# B&R Automation Studio project CombinedLinenCleanA6 (part 7)

#### _SetCAN2TypeToCAN1Type.ab
```automation-basic
FUNCTION_BLOCK _SetCAN2TypeToCAN1Type
;********************************************************************************************************
; * Implementation of _SetCAN2TypeToCAN1Type
;********************************************************************************************************
; * version 		1.10
;	* ###HO - 020905 - Fünftes Telegramm ergänzt
; * version 		1.00
; * last change		sep, 30th, 2003
; * by				H.O.
;********************************************************************************************************
;********************************************************************************************************
; 	-> 	pCAN2Data			.. pointer to CAN2 structure that contains data to read or write
; 	-> 	iTelegramIndex		.. telegram index exctractet from received / broadcasted telegram
; 		pCAN1Data 		->	.. return the address of CAN1 struct
;********************************************************************************************************

; set local pointer to incoming CAN2 uni structure
memcpy(adr(LocalCAN2UniData), pCAN2Data, sizeof(LocalCAN2UniData))

iStatus = 0

; create CAN1 telegram from CAN2 te structure passed in..
case iTelegramIndex of
	action 1:
		LocalCAN1Data.T_By0 	= LocalCAN2UniData.T1_By0
		LocalCAN1Data.T_By1 	= LocalCAN2UniData.T1_By1
		LocalCAN1Data.T_By2_By3 = LocalCAN2UniData.T1_By2_By3
		LocalCAN1Data.T_By4_By5 = LocalCAN2UniData.T1_By4_By5
		LocalCAN1Data.T_By6_By7 = LocalCAN2UniData.T1_By6_By7
	endaction
	action 2:
		LocalCAN1Data.T_By0 	= LocalCAN2UniData.T2_By0
		LocalCAN1Data.T_By1 	= LocalCAN2UniData.T2_By1
		LocalCAN1Data.T_By2_By3 = LocalCAN2UniData.T2_By2_By3
		LocalCAN1Data.T_By4_By5 = LocalCAN2UniData.T2_By4_By5
		LocalCAN1Data.T_By6_By7 = LocalCAN2UniData.T2_By6_By7
	endaction
	action 3:
		LocalCAN1Data.T_By0 	= LocalCAN2UniData.T3_By0
		LocalCAN1Data.T_By1 	= LocalCAN2UniData.T3_By1
		LocalCAN1Data.T_By2_By3 = LocalCAN2UniData.T3_By2_By3
		LocalCAN1Data.T_By4_By5 = LocalCAN2UniData.T3_By4_By5
		LocalCAN1Data.T_By6_By7 = LocalCAN2UniData.T3_By6_By7
	endaction
	action 4:
		LocalCAN1Data.T_By0 	= LocalCAN2UniData.T4_By0
		LocalCAN1Data.T_By1 	= LocalCAN2UniData.T4_By1
		LocalCAN1Data.T_By2_By3 = LocalCAN2UniData.T4_By2_By3
		LocalCAN1Data.T_By4_By5 = LocalCAN2UniData.T4_By4_By5
		LocalCAN1Data.T_By6_By7 = LocalCAN2UniData.T4_By6_By7
	endaction
	action 5:
		LocalCAN1Data.T_By0 	= LocalCAN2UniData.T5_By0
		LocalCAN1Data.T_By1 	= LocalCAN2UniData.T5_By1
		LocalCAN1Data.T_By2_By3 = LocalCAN2UniData.T5_By2_By3
		LocalCAN1Data.T_By4_By5 = LocalCAN2UniData.T5_By4_By5
		LocalCAN1Data.T_By6_By7 = LocalCAN2UniData.T5_By6_By7
	endaction
	elseaction:
		iStatus = 109
	endaction
endcase

; pass pointer to CAN1 telegram to output..
pCAN1Data = ADR(LocalCAN1Data)

;********************************************************************************************************
;********************************************************************************************************
END_FUNCTION_BLOCK
```

#### _GetCANIDFromObjNr.ab
```automation-basic
FUNCTION_BLOCK _GetCANIDFromObjNr
;********************************************************************************************************
; * Implementation of _GetCANIDFromObjNr
;********************************************************************************************************
; * version 		3.6.0
; * last change		120210
; * by				H.O.
;********************************************************************************************************
; History:
;*********
; V3.6.0 - ###HO - 120210
;	* COB120 auch für ID 150,160,170,180,190
;	* COB121 auch für ID 151,161,171,181,191
; * V3.4.0 ###HO
; 	- COB ID 110 + 111
; * V3.2.1 ###HO
; 	- COB 130,140 wie 120  und...
;	- 131 und 141 wie 121
; * V3.2.0 ###HO  - 040907
;  	* COBs 261+262 hinzugefügt
; 	* COBs302,303,304,312,313,314,253,255,254,256,352,353,354  neu
;	* udCANID = udObjNr für alle erwähnten Objektnummern
; * V3.1.0 ###HO  - 141206
; 	* COBs 126,127,128,129 hinzugefügt
; * V3.0.0 ###HO  - 120905
; 	* IDs 253..258 hinzugefügt
; 	* IDs 307..317 hinzugefügt
; * V 1.0.0  	* Erste Version
; * V 2.0.0 HO 	* COBs 251,252,480,481 added
; 				* COB 123 added
; * V2.1.0 HO	* COB 441..459 added
;********************************************************************************************************
; supported CANIDs: 120,121,122,123,130,140,131,141,201,209,211,219,221,231,251,252
; 					301,306,311,316,351,361..369,371..379,401..419,421..439,441..459,480,481
;********************************************************************************************************

; ObjNr and CANID are identical..
iStatus = 0
case udObjNr of

    action 120 :
    action 126 :
    action 128 :
    action 130 :
    action 140 :
	action 150:
	action 160:
	action 170:
	action 180:
	action 190:
        udCANID = 120
    endaction
   	action 121:
    action 127 :
    action 129 :
    action 131 :
    action 141 :
	action 151:
	action 161:
	action 171:
	action 181:
	action 191:
        udCANID = 121
	endaction

	action 110 :
	action 111 :
	action 122 :
   	action 123 :
	action 201:
	action 209:
	action 211:
	action 219:
	action 221:
	action 231:
	action 251:
	action 252:
	action 253:
	action 254:
	action 255:
	action 256:
	action 257:
	action 258:
	action 261:
	action 262:
	action 301:
	action 302:
	action 303:
	action 304:
	action 306:
	action 307:
	action 311:
	action 312:
	action 313:
	action 314:
	action 316:
	action 317:
	action 351:
	action 352:
	action 353:
	action 354:
	action 361..369:
	action 371..379:
	action 401..419:
	action 421..439:
	action 441..459:
	action 480:
	action 481:
        udCANID = udObjNr
	endaction
	elseaction:
		; all other ObjNrs..
		iStatus = 110
	endaction
endcase
;********************************************************************************************************
END_FUNCTION_BLOCK
```

#### _GetPVSize.ab
```automation-basic
FUNCTION_BLOCK _GetPVSize
;********************************************************************************************************
; * Implementation of _GetPVSize
;********************************************************************************************************
; * version 		3.6.0
; * last change		120210
; * by				H.O.
;********************************************************************************************************
; History:
;*********
; V3.6.0 - ###HO - 120210
;	* COB120 auch für ID 150,160,170,180,190
;	* COB121 auch für ID 151,161,171,181,191
; * V3.4.0
;	* COB ID 110 + 111
; * V3.2.1
;	* COB130,140 wie 120 und..
;	* COB 131,141 wie 121
; * V3.2.0
; 	* COBs 261,262 hinzugefügt
; 	* COBs302,303,304,312,313,314,253,255,254,256,352,353,354  neu
; 	* gleiche Objekte durch MehrfachAction zusammengefasst
; * V3.1.0
; 	* COBs 126,127,128,129,130 hinzugefügt
; * V3.0.0
; 	* COBs 253..258 -> gleiche Strukturen mit anderen IDs (hcs)
; * V 1.0.0 	-> Original
; * V 2.0.0 HO 	* COBs 251,252,480,481 added
;				* COB 123 added
; * V2.1.0	HO	* COB441..459 added

;********************************************************************************************************
; supported CANIDs: 120,121,122,123,130,140,131,141,201,209,211,219,221,231,251,252
; 					301,306,311,316,351,361..369,371..379,401..419,421..439,441bis459,480,481
;********************************************************************************************************

iStatus = 0
case uiObjNr of
action 110:
	iCobLength = sizeof (COB_Typ_110)
endaction
action 111:
	iCobLength = sizeof (COB_Typ_111)
endaction
action 120:
action 126:
action 128:
action 130:
action 140:
action 150:
action 160:
action 170:
action 180:
action 190:
	iCobLength = sizeof (COBTyp_120)
endaction
action 121:
action 127:
action 129:
action 131:
action 141:
action 151:
action 161:
action 171:
action 181:
action 191:
	iCobLength = sizeof (COBTyp_121)
endaction
action 122:
	iCobLength = sizeof (COBTyp_122)
endaction
action 123:
	iCobLength = sizeof (COBTyp_123)
endaction
(*
action 1130:	; 08.10.2007 - (hcs) DEAKTIVIERT
	iCobLength = sizeof (COB_Typ_130_140)
endaction
action 1131:	; 08.10.2007 - (hcs) DEAKTIVIERT
  	iCobLength = sizeof (COB_Typ_131_141)
endaction
action 140:
	iCobLength = sizeof (COB_Typ_130_140)
endaction
action 141:
  	iCobLength = sizeof (COB_Typ_131_141)
endaction
*)
action 201:
   	iCobLength = sizeof (COB_Typ_201)
endaction
action 209:
   	iCobLength = sizeof (COB_Typ_209)
endaction
action 211:
   	iCobLength = sizeof (COB_Typ_211)
endaction
action 219:
   	iCobLength = sizeof (COB_Typ_219)
endaction
action 221:
	iCobLength = sizeof (COB_Typ_221)
endaction
action 231:
	iCobLength = sizeof (COB_Typ_231)
endaction
action 251:
action 253:
action 255:
action 257:
	iCobLength = sizeof (COBTyp_251)
endaction
action 252:
action 254:
action 256:
action 258:
	iCobLength = sizeof (COBTyp_252)
endaction
action 261:
	iCobLength = sizeof (COB_Typ_261)
endaction
action 262:
	iCobLength = sizeof (COB_Typ_262)
endaction
action 301:
action 302:
action 303:
action 304:
	iCobLength = sizeof (COB_Typ_301)
endaction
action 306:
	iCobLength = sizeof (COB_Typ_306)
endaction
action 307:
	iCobLength = sizeof (COB_Typ_307)
endaction
action 311:
action 312:
action 313:
action 314:
	iCobLength = sizeof (COB_Typ_311)
endaction
action 316:
	iCobLength = sizeof (COB_Typ_316)
endaction
action 317:
	iCobLength = sizeof (COB_Typ_317)
endaction
action 351:
action 352:
action 353:
action 354:
	iCobLength = sizeof (COB_Typ_351)
endaction
action 361..369:
	iCobLength = sizeof (COB_Typ_361bis369)
endaction
action 371..379:
	iCobLength = sizeof (COB_Typ_371bis379)
endaction
action 401..419:
	iCobLength = sizeof (COB_Typ_401bis419)
endaction
action 421..439:
	iCobLength = sizeof (COB_Typ_421bis439)
endaction
action 441..459:
	iCobLength = sizeof (COB_Typ_441bis459)
endaction
action 480:
	iCobLength = sizeof (COBTyp_480)
endaction
action 481:
	iCobLength = sizeof (COBTyp_481)
endaction

; all other ObjNrs..
elseaction:
	iStatus = 110
endaction

endcase
;********************************************************************************************************
END_FUNCTION_BLOCK
```

#### _ConvertDataToi386.ab
```automation-basic
FUNCTION_BLOCK _ConvertDataToi386
;********************************************************************************************************
; * Implementation of _ConvertDataToi386
; 	*** Only ReadOperation for IntelTarget***
;********************************************************************************************************
; * version 		3.6.0
; * last change		120210
; * by				H.O.
;********************************************************************************************************
; History:
; --------
; V3.6.0 - ###HO - 120210
;	* COB120 auch für ID 150,160,170,180,190
;	* COB121 auch für ID 151,161,171,181,191
; * V3.4.0
;	* COB ID 110 + 111
; * V3.2.1
;	* COB130,140 wie 120 und..
;	* COB 131,141 wie 121
; * V3.2.0 HO 040907
;	* _ConvertDataToi386.COB251.bStartBeladung
;	* COBs 261,262 added
; 	* COBs302,303,304,312,313,314,253,255,254,256,352,353,354  neu
; * V3.1.0 HO 141206
;	* COBs 126,127,128,129 hinzugefügt
; * V3.0.0 HO 070905
;		cob251
; * V2.1.0 HO 150404
;		* Redundancy support done for COBs: 480,481
; * V 2.0.0 (by HO) -> COBs 251,252,480,481 added
; 					-> COBs 120,121,123 modified
; 					-> COB 122 replaced
; * V 1.0.0  		-> Original
;********************************************************************************************************
; this function transforms an incoming ByteArray in motorola order to intel format:
;  -> performs address adaption to intel format
; 		(intel requires swapping of WORDs and modification of startadresses by DWORDs (dividable by four))
;  -> swapping of single WORDS of LONG
;  -> swapping of single WORDS (= uints) is not necessary
;  -> swapping of neighboring characters of STRING
;********************************************************************************************************
; supported CANIDs: 120, 121,122,123,130,140,131,141,201,209,211,219,221,231,251,252
; 					301,306,311,316,351,361..369,371..379,401..419,421..439,480,481
;********************************************************************************************************

; always assign InData to OutData -> overwrite changes..
ByteArrayi386 = ByteArrayMotorola

case uiObjNr of
	action 120:
	action 126:
	action 128:
	action 130:
	action 140:
	action 150:
	action 160:
	action 170:
	action 180:
	action 190:
		; udPostennummer
		ByteArrayi386[8] 	= ByteArrayMotorola[10]
		ByteArrayi386[9] 	= ByteArrayMotorola[11]
		ByteArrayi386[10] 	= ByteArrayMotorola[8]
		ByteArrayi386[11] 	= ByteArrayMotorola[9]

		; szAuftragskennzeichen
		usTempByte 			= ByteArrayMotorola[14]
		ByteArrayi386[14] 	= ByteArrayMotorola[15]
		ByteArrayi386[15] 	= usTempByte
		usTempByte 			= ByteArrayMotorola[16]
		ByteArrayi386[16] 	= ByteArrayMotorola[17]
		ByteArrayi386[17] 	= usTempByte
		usTempByte 			= ByteArrayMotorola[18]
		ByteArrayi386[18] 	= ByteArrayMotorola[19]
		ByteArrayi386[19] 	= usTempByte
		usTempByte 			= ByteArrayMotorola[20]
		ByteArrayi386[20] 	= ByteArrayMotorola[21]
		ByteArrayi386[21] 	= usTempByte
		usTempByte 			= ByteArrayMotorola[22]
		ByteArrayi386[22] 	= ByteArrayMotorola[23]
		ByteArrayi386[23] 	= usTempByte
		usTempByte 			= ByteArrayMotorola[24]
		ByteArrayi386[24] 	= ByteArrayMotorola[25]
		ByteArrayi386[25] 	= usTempByte
		; + EOS +  Alignment

		; ud Kundennummer
		ByteArrayi386[28] 	= ByteArrayMotorola[30]
		ByteArrayi386[29] 	= ByteArrayMotorola[31]
		ByteArrayi386[30] 	= ByteArrayMotorola[28]
		ByteArrayi386[31] 	= ByteArrayMotorola[29]

	endaction ; 120

	action 121:
	action 127:
	action 129:
	action 131:
	action 141:
	action 151:
	action 161:
	action 171:
	action 181:
	action 191:
		; nothing to do..
	endaction ; 121

	; replaced from V2.0.0
	action 122:
		; udKundennummer
		ByteArrayi386[4] 	= ByteArrayMotorola[6]
		ByteArrayi386[5] 	= ByteArrayMotorola[7]
		ByteArrayi386[6] 	= ByteArrayMotorola[4]
		ByteArrayi386[7] 	= ByteArrayMotorola[5]

		; udPostennummer
		ByteArrayi386[12] 	= ByteArrayMotorola[14]
		ByteArrayi386[13] 	= ByteArrayMotorola[15]
		ByteArrayi386[14] 	= ByteArrayMotorola[12]
		ByteArrayi386[15] 	= ByteArrayMotorola[13]

		; szAuftragskennzeichen
		usTempByte 			= ByteArrayMotorola[17]
		ByteArrayi386[17] 	= ByteArrayMotorola[18]
		ByteArrayi386[18] 	= usTempByte
		usTempByte 			= ByteArrayMotorola[19]
		ByteArrayi386[19] 	= ByteArrayMotorola[20]
		ByteArrayi386[20] 	= usTempByte
		usTempByte 			= ByteArrayMotorola[21]
		ByteArrayi386[21] 	= ByteArrayMotorola[22]
		ByteArrayi386[22] 	= usTempByte
		usTempByte 			= ByteArrayMotorola[23]
		ByteArrayi386[23] 	= ByteArrayMotorola[24]
		ByteArrayi386[24] 	= usTempByte
		usTempByte 			= ByteArrayMotorola[25]
		ByteArrayi386[25] 	= ByteArrayMotorola[26]
		ByteArrayi386[26] 	= usTempByte
		usTempByte 			= ByteArrayMotorola[27]
		ByteArrayi386[27] 	= ByteArrayMotorola[28]
		ByteArrayi386[28] 	= usTempByte
	endaction ; 122

	action 123:
		; nothing to do..
	endaction ; 123
(*
	action 1130: 			; 08.10.2007 - (hcs) DEAKTIVIERT
		; udPostennummer
		ByteArrayi386[12] 	= ByteArrayMotorola[12]
		ByteArrayi386[13] 	= ByteArrayMotorola[13]
		ByteArrayi386[14] 	= ByteArrayMotorola[10]
		ByteArrayi386[15] 	= ByteArrayMotorola[11]

		; usFehlernummer
		ByteArrayi386[16] 	= ByteArrayMotorola[14]

		; bAuftragskennzeichen
		ByteArrayi386[17] 	= ByteArrayMotorola[15]

		; szAuftragskennzeichen
			ByteArrayi386[18] 	= ByteArrayMotorola[17]
		ByteArrayi386[19] 	= ByteArrayMotorola[16]
			ByteArrayi386[20] 	= ByteArrayMotorola[19]
		ByteArrayi386[21] 	= ByteArrayMotorola[18]
			ByteArrayi386[22] 	= ByteArrayMotorola[21]
		ByteArrayi386[23] 	= ByteArrayMotorola[20]
			ByteArrayi386[24] 	= ByteArrayMotorola[23]
		ByteArrayi386[25] 	= ByteArrayMotorola[22]
			ByteArrayi386[26] 	= ByteArrayMotorola[25]
		ByteArrayi386[27] 	= ByteArrayMotorola[24]
			ByteArrayi386[28] 	= ByteArrayMotorola[27]
		ByteArrayi386[29] 	= ByteArrayMotorola[26]

		; udKundennummer
		ByteArrayi386[32] 	= ByteArrayMotorola[32]
		ByteArrayi386[33] 	= ByteArrayMotorola[33]
		ByteArrayi386[34] 	= ByteArrayMotorola[30]
		ByteArrayi386[35] 	= ByteArrayMotorola[31]

		; uiGewicht
		ByteArrayi386[36] 	= ByteArrayMotorola[34]
		ByteArrayi386[37] 	= ByteArrayMotorola[35]

		; bNotAusEnts
		ByteArrayi386[38] 	= ByteArrayMotorola[36]
	endaction ; 130

	action 140:
		; udPostennummer
		ByteArrayi386[12] 	= ByteArrayMotorola[12]
		ByteArrayi386[13] 	= ByteArrayMotorola[13]
		ByteArrayi386[14] 	= ByteArrayMotorola[10]
		ByteArrayi386[15] 	= ByteArrayMotorola[11]

		; usFehlernummer
		ByteArrayi386[16] 	= ByteArrayMotorola[14]

		; bAuftragskennzeichen
		ByteArrayi386[17] 	= ByteArrayMotorola[15]

		; szAuftragskennzeichen
			ByteArrayi386[18] 	= ByteArrayMotorola[17]
		ByteArrayi386[19] 	= ByteArrayMotorola[16]
			ByteArrayi386[20] 	= ByteArrayMotorola[19]
		ByteArrayi386[21] 	= ByteArrayMotorola[18]
			ByteArrayi386[22] 	= ByteArrayMotorola[21]
		ByteArrayi386[23] 	= ByteArrayMotorola[20]
			ByteArrayi386[24] 	= ByteArrayMotorola[23]
		ByteArrayi386[25] 	= ByteArrayMotorola[22]
			ByteArrayi386[26] 	= ByteArrayMotorola[25]
		ByteArrayi386[27] 	= ByteArrayMotorola[24]
			ByteArrayi386[28] 	= ByteArrayMotorola[27]
		ByteArrayi386[29] 	= ByteArrayMotorola[26]

		; udKundennummer
		ByteArrayi386[32] 	= ByteArrayMotorola[32]
		ByteArrayi386[33] 	= ByteArrayMotorola[33]
		ByteArrayi386[34] 	= ByteArrayMotorola[30]
		ByteArrayi386[35] 	= ByteArrayMotorola[31]

		; uiGewicht
		ByteArrayi386[36] 	= ByteArrayMotorola[34]
		ByteArrayi386[37] 	= ByteArrayMotorola[35]

		; bNotAusEnts
		ByteArrayi386[38] 	= ByteArrayMotorola[36]
	endaction ; 140

	action 1131: 	; 08.10.2007 - (hcs) DEAKTIVIERT
		; nothing to do
	endaction ; 131..141

	action 141:
		; nothing to do
	endaction ; 131..141
*)
	action 201:
	; nur swappen - kein Alignment
		; udPostennummer
		ByteArrayi386[8] 	= ByteArrayMotorola[10]
		ByteArrayi386[9] 	= ByteArrayMotorola[11]
		ByteArrayi386[10] 	= ByteArrayMotorola[8]
		ByteArrayi386[11] 	= ByteArrayMotorola[9]

		; udKundennummer
		ByteArrayi386[12] 	= ByteArrayMotorola[14]
		ByteArrayi386[13] 	= ByteArrayMotorola[15]
		ByteArrayi386[14] 	= ByteArrayMotorola[12]
		ByteArrayi386[15] 	= ByteArrayMotorola[13]
	endaction ; 201

	action 209:
		; udPostennummer
		ByteArrayi386[8] 	= ByteArrayMotorola[10]
		ByteArrayi386[9] 	= ByteArrayMotorola[11]
		ByteArrayi386[10] 	= ByteArrayMotorola[8]
		ByteArrayi386[11] 	= ByteArrayMotorola[9]

		; udKundennummer
		ByteArrayi386[12] 	= ByteArrayMotorola[14]
		ByteArrayi386[13] 	= ByteArrayMotorola[15]
		ByteArrayi386[14] 	= ByteArrayMotorola[12]
		ByteArrayi386[15] 	= ByteArrayMotorola[13]
	endaction ; 209

	action 211:
		; nothing to do
	endaction ; 211

	action 219:
		; nothing to do
		ByteArrayi386[6] 	= ByteArrayMotorola[7]
		ByteArrayi386[7] 	= ByteArrayMotorola[6]
	endaction ; 219

	action 221:
		; udPostennummer
		ByteArrayi386[8] 	= ByteArrayMotorola[8]
		ByteArrayi386[9] 	= ByteArrayMotorola[9]
		ByteArrayi386[10] 	= ByteArrayMotorola[6]
		ByteArrayi386[11] 	= ByteArrayMotorola[7]
		; udKundennummer
		ByteArrayi386[12] 	= ByteArrayMotorola[12]
		ByteArrayi386[13] 	= ByteArrayMotorola[13]
		ByteArrayi386[14] 	= ByteArrayMotorola[10]
		ByteArrayi386[15] 	= ByteArrayMotorola[11]
		; uiGewicht
		ByteArrayi386[16] 	= ByteArrayMotorola[14]
		ByteArrayi386[17] 	= ByteArrayMotorola[15]
		; bNotAusWM
		ByteArrayi386[18] 	= ByteArrayMotorola[16]
		; Res
		ByteArrayi386[19] 	= ByteArrayMotorola[17]
		ByteArrayi386[20] 	= ByteArrayMotorola[18]
		; a_usCustomize
		ByteArrayi386[21] 	= ByteArrayMotorola[19]
		ByteArrayi386[22] 	= ByteArrayMotorola[20]
		ByteArrayi386[23] 	= ByteArrayMotorola[21]
		ByteArrayi386[24] 	= ByteArrayMotorola[22]
		ByteArrayi386[25] 	= ByteArrayMotorola[23]
		ByteArrayi386[26] 	= ByteArrayMotorola[24]
		ByteArrayi386[27] 	= ByteArrayMotorola[25]
	endaction ; 221

	action 231:
		; nothing to do
	endaction ; 231
	action 251:
	action 253:
	action 255:
	action 257:
		; udPostennummer
		ByteArrayi386[8] 	= ByteArrayMotorola[8]
		ByteArrayi386[9] 	= ByteArrayMotorola[9]
		ByteArrayi386[10] 	= ByteArrayMotorola[6]
		ByteArrayi386[11] 	= ByteArrayMotorola[7]

		; udKundennummer
		ByteArrayi386[12] 	= ByteArrayMotorola[12]
		ByteArrayi386[13] 	= ByteArrayMotorola[13]
		ByteArrayi386[14] 	= ByteArrayMotorola[10]
		ByteArrayi386[15] 	= ByteArrayMotorola[11]

		; uiGewicht
		ByteArrayi386[16] 	= ByteArrayMotorola[14]
		ByteArrayi386[17] 	= ByteArrayMotorola[15]

		; usZiel
		ByteArrayi386[18] 	= ByteArrayMotorola[16]

		; bBeladeende
		ByteArrayi386[19] 	= ByteArrayMotorola[17]

		; usReserve
		ByteArrayi386[20] 	= ByteArrayMotorola[18]

		; bSperreBereich
		ByteArrayi386[21] 	= ByteArrayMotorola[19]

		; a_usCustomize
		ByteArrayi386[22] 	= ByteArrayMotorola[20]
		ByteArrayi386[23] 	= ByteArrayMotorola[21]
		ByteArrayi386[24] 	= ByteArrayMotorola[22]
		ByteArrayi386[25] 	= ByteArrayMotorola[23]
		ByteArrayi386[26] 	= ByteArrayMotorola[24]
		ByteArrayi386[27] 	= ByteArrayMotorola[25]
		ByteArrayi386[28] 	= ByteArrayMotorola[26]

		; bStartBeladung	###HO - 040907
		ByteArrayi386[29] 	= ByteArrayMotorola[27]

	endaction ; 251

	action 252:
	action 254:
	action 256:
	action 258:
		; nothing to do..
	endaction ; 252

	action 261:
		; nothing to do..
	endaction ; 261
	action 262:
		; nothing to do..
	endaction ; 262

	action 301:
	action 302:
	action 303:
	action 304:
		; udPostennummer
		ByteArrayi386[8] 	= ByteArrayMotorola[10]
		ByteArrayi386[9] 	= ByteArrayMotorola[11]
		ByteArrayi386[10] 	= ByteArrayMotorola[8]
		ByteArrayi386[11] 	= ByteArrayMotorola[9]

		; udKundennummer
		ByteArrayi386[12] 	= ByteArrayMotorola[14]
		ByteArrayi386[13] 	= ByteArrayMotorola[15]
		ByteArrayi386[14] 	= ByteArrayMotorola[12]
		ByteArrayi386[15] 	= ByteArrayMotorola[13]
	endaction ; 301

;	action 110:
	action 306:
		; udPostennummer
		ByteArrayi386[8] 	= ByteArrayMotorola[10]
		ByteArrayi386[9] 	= ByteArrayMotorola[11]
		ByteArrayi386[10] 	= ByteArrayMotorola[8]
		ByteArrayi386[11] 	= ByteArrayMotorola[9]

		; udKundennummer
		ByteArrayi386[12] 	= ByteArrayMotorola[14]
		ByteArrayi386[13] 	= ByteArrayMotorola[15]
		ByteArrayi386[14] 	= ByteArrayMotorola[12]
		ByteArrayi386[15] 	= ByteArrayMotorola[13]
	endaction ; 306

	action 307:
		; udPostennummer
		ByteArrayi386[8] 	= ByteArrayMotorola[10]
		ByteArrayi386[9] 	= ByteArrayMotorola[11]
		ByteArrayi386[10] 	= ByteArrayMotorola[8]
		ByteArrayi386[11] 	= ByteArrayMotorola[9]

		; udKundennummer
		ByteArrayi386[16] 	= ByteArrayMotorola[18]
		ByteArrayi386[17] 	= ByteArrayMotorola[19]
		ByteArrayi386[18] 	= ByteArrayMotorola[16]
		ByteArrayi386[19] 	= ByteArrayMotorola[17]
	endaction ; 307

	action 311:
	action 312:
	action 313:
	action 314:
		; nothing to do
	endaction ; 311

	action 111:
	action 316:
		; nothing to do
	endaction ; 316

	action 351:
	action 352:
	action 353:
	action 354:
		; udPostennummer
		ByteArrayi386[8] 	= ByteArrayMotorola[10]
		ByteArrayi386[9] 	= ByteArrayMotorola[11]
		ByteArrayi386[10] 	= ByteArrayMotorola[8]
		ByteArrayi386[11] 	= ByteArrayMotorola[9]

		; udKundennummer
		ByteArrayi386[12] 	= ByteArrayMotorola[14]
		ByteArrayi386[13] 	= ByteArrayMotorola[15]
		ByteArrayi386[14] 	= ByteArrayMotorola[12]
		ByteArrayi386[15] 	= ByteArrayMotorola[13]
	endaction ; 351

	action 361..369:
		; udPostennummer
		ByteArrayi386[4] 	= ByteArrayMotorola[6]
		ByteArrayi386[5] 	= ByteArrayMotorola[7]
		ByteArrayi386[6] 	= ByteArrayMotorola[4]
		ByteArrayi386[7] 	= ByteArrayMotorola[5]

		; udKundennummer
		ByteArrayi386[8] 	= ByteArrayMotorola[10]
		ByteArrayi386[9] 	= ByteArrayMotorola[11]
		ByteArrayi386[10] 	= ByteArrayMotorola[8]
		ByteArrayi386[11] 	= ByteArrayMotorola[9]
	endaction ; 361..369

	action 371..379:
		; nothing to do
	endaction ; 371..379

	action 401..419:
		; udPostennummer
		ByteArrayi386[8] 	= ByteArrayMotorola[10]
		ByteArrayi386[9] 	= ByteArrayMotorola[11]
		ByteArrayi386[10] 	= ByteArrayMotorola[8]
		ByteArrayi386[11] 	= ByteArrayMotorola[9]

		; udKundennummer
		ByteArrayi386[12] 	= ByteArrayMotorola[14]
		ByteArrayi386[13] 	= ByteArrayMotorola[15]
		ByteArrayi386[14] 	= ByteArrayMotorola[12]
		ByteArrayi386[15] 	= ByteArrayMotorola[13]
	endaction ; 401..419

	action 421..439:
		; uszuluftTemp + usAbluftIRTemp
		ByteArrayi386[12] 	= ByteArrayMotorola[13]
		ByteArrayi386[13] 	= ByteArrayMotorola[12]
		; udPostennummer
		ByteArrayi386[24] 	= ByteArrayMotorola[24]
		ByteArrayi386[25] 	= ByteArrayMotorola[25]
		ByteArrayi386[26] 	= ByteArrayMotorola[22]
		ByteArrayi386[27] 	= ByteArrayMotorola[23]
		; udKundennummer
		ByteArrayi386[28] 	= ByteArrayMotorola[28]
		ByteArrayi386[29] 	= ByteArrayMotorola[29]
		ByteArrayi386[30] 	= ByteArrayMotorola[26]
		ByteArrayi386[31] 	= ByteArrayMotorola[27]
		; uiGewicht
		ByteArrayi386[32] 	= ByteArrayMotorola[30]
		ByteArrayi386[33] 	= ByteArrayMotorola[31]
		; bNotAusTrockner
		ByteArrayi386[34] 	= ByteArrayMotorola[32]
		; bHand
		ByteArrayi386[35] 	= ByteArrayMotorola[33]
		; uiIRTemp
		ByteArrayi386[37] 	= ByteArrayMotorola[34]
		ByteArrayi386[36] 	= ByteArrayMotorola[35]
		; usReserve
		ByteArrayi386[38] 	= ByteArrayMotorola[36]
		; a_usCustomize
		ByteArrayi386[39] 	= ByteArrayMotorola[37]
		ByteArrayi386[40] 	= ByteArrayMotorola[38]
		ByteArrayi386[41] 	= ByteArrayMotorola[39]
		ByteArrayi386[42] 	= ByteArrayMotorola[40]
		ByteArrayi386[43] 	= ByteArrayMotorola[41]
		ByteArrayi386[44] 	= ByteArrayMotorola[42]
		ByteArrayi386[45] 	= ByteArrayMotorola[43]
	endaction ; 421..439

	action 480:
		; udPostennummer
		ByteArrayi386[16] 	= ByteArrayMotorola[16]
		ByteArrayi386[17] 	= ByteArrayMotorola[17]
		ByteArrayi386[18] 	= ByteArrayMotorola[14]
		ByteArrayi386[19] 	= ByteArrayMotorola[15]
		; udKundennummer
		ByteArrayi386[20] 	= ByteArrayMotorola[20]
		ByteArrayi386[21] 	= ByteArrayMotorola[21]
		ByteArrayi386[22] 	= ByteArrayMotorola[18]
		ByteArrayi386[23] 	= ByteArrayMotorola[19]
		; uiGewicht
		ByteArrayi386[24] 	= ByteArrayMotorola[22]
		ByteArrayi386[25] 	= ByteArrayMotorola[23]
		; usReserve1
		ByteArrayi386[26] 	= ByteArrayMotorola[24]
		;bReserve1-bReserve9
		ByteArrayi386[27] 	= ByteArrayMotorola[25]
		ByteArrayi386[28] 	= ByteArrayMotorola[26]
		ByteArrayi386[29] 	= ByteArrayMotorola[27]
		ByteArrayi386[30] 	= ByteArrayMotorola[28]
		ByteArrayi386[31] 	= ByteArrayMotorola[29]
		ByteArrayi386[32] 	= ByteArrayMotorola[30]
		ByteArrayi386[33] 	= ByteArrayMotorola[31]
		ByteArrayi386[34] 	= ByteArrayMotorola[32]
		ByteArrayi386[35] 	= ByteArrayMotorola[33]
		; a_usCustomize
		ByteArrayi386[36] 	= ByteArrayMotorola[34]
		ByteArrayi386[37] 	= ByteArrayMotorola[35]
		ByteArrayi386[38] 	= ByteArrayMotorola[36]
		ByteArrayi386[39] 	= ByteArrayMotorola[37]
		ByteArrayi386[40] 	= ByteArrayMotorola[38]
		ByteArrayi386[41] 	= ByteArrayMotorola[39]
		ByteArrayi386[42] 	= ByteArrayMotorola[40]
	endaction ; 480

	action 481:
		; udKundennummer
		ByteArrayi386[16] 	= ByteArrayMotorola[16]
		ByteArrayi386[17] 	= ByteArrayMotorola[17]
		ByteArrayi386[18] 	= ByteArrayMotorola[14]
		ByteArrayi386[19] 	= ByteArrayMotorola[15]
		; udPostennummer
		ByteArrayi386[20] 	= ByteArrayMotorola[20]
		ByteArrayi386[21] 	= ByteArrayMotorola[21]
		ByteArrayi386[22] 	= ByteArrayMotorola[18]
		ByteArrayi386[23] 	= ByteArrayMotorola[19]
		; usReserve1
		ByteArrayi386[24] 	= ByteArrayMotorola[22]
		;bReserve1-bReserve10
		ByteArrayi386[25] 	= ByteArrayMotorola[23]
		ByteArrayi386[26] 	= ByteArrayMotorola[24]
		ByteArrayi386[27] 	= ByteArrayMotorola[25]
		ByteArrayi386[28] 	= ByteArrayMotorola[26]
		ByteArrayi386[29] 	= ByteArrayMotorola[27]
		ByteArrayi386[30] 	= ByteArrayMotorola[28]
		ByteArrayi386[31] 	= ByteArrayMotorola[29]
		ByteArrayi386[32] 	= ByteArrayMotorola[30]
		ByteArrayi386[33] 	= ByteArrayMotorola[31]
		ByteArrayi386[34] 	= ByteArrayMotorola[32]
		; a_usCustomize
		ByteArrayi386[35] 	= ByteArrayMotorola[33]
		ByteArrayi386[36] 	= ByteArrayMotorola[34]
		ByteArrayi386[37] 	= ByteArrayMotorola[35]
		ByteArrayi386[38] 	= ByteArrayMotorola[36]
		ByteArrayi386[39] 	= ByteArrayMotorola[37]
		ByteArrayi386[40] 	= ByteArrayMotorola[38]
		ByteArrayi386[41] 	= ByteArrayMotorola[39]
	endaction ; 481
endcase

;******************************************************************
END_FUNCTION_BLOCK
```

- Data object Logical/ioimgcfg (Simple) (no source held here)

### Data object Logical/a_flx_io (Simple)

#### a_flx_io.dat
```
; Automation Studio generated file.
; Each change of the file content causes the deactivation
; of the further automatic actualization of this file by the Automation Studio!

"IDP5.0.05.01, X301, TC#2i"
"IDP5.0.05.02, X302, TC#2i"
"IDP5.0.05.03, X303, TC#2i"
"IDP5.0.05.05, X305, TC#2i"
"IDP5.0.05.06, X306, TC#2i"
"IDP5.0.05.07, X307, TC#2i"
"IDP5.0.05.08, X308, TC#2i"
"IDP5.0.05.09, X309, TC#2i"
"IDP5.0.05.10, X310, TC#2i"
"IDP5.0.05.11, X311, TC#2i"
"IDP5.0.05.12, X312, TC#2i"
"IDP5.0.05.13, X313, TC#2i"
"IDP5.0.05.14, X314, TC#2i"
"IDP5.0.05.15, X315, TC#2i"
"IDP5.0.05.16, X316, TC#2i"
"IDP5.0.06.01, X401, TC#2i"
"IDP5.0.06.02, X402, TC#2i"
"IDP5.0.06.03, X403, TC#2i"
"IDP5.0.06.04, X404, TC#2i"
"IDP5.0.06.05, X405, TC#2i"
"IDP5.0.06.06, X406, TC#2i"
"IDP5.0.06.08, X408, TC#2i"
"IDP5.0.06.10, X410, TC#2i"
"IDP5.0.06.12, X412, TC#2i"
"IDP5.0.06.13, X413, TC#2i"
"IDP5.0.06.14, X414, TC#2i"
"IDP5.0.06.15, X415, TC#2i"
"IDP5.0.07.01, X501, TC#2i"
"IDP5.0.07.02, X502, TC#2i"
"IDP5.0.07.03, X503, TC#2i"
"IDP5.0.07.04, X504, TC#2i"
"IDP5.0.07.05, X505, TC#2i"
"IDP5.0.07.06, X506, TC#2i"
"IDP5.0.07.09, X509, TC#2i"
"IDP5.0.07.10, X510, TC#2i"
"IDP5.0.07.12, X512, TC#2i"
"IDP5.0.07.13, X513, TC#2i"
"IDP5.0.07.14, X514, TC#2i"
"IDP5.0.07.15, X515, TC#2i"
"IDP5.0.08.03, X603, TC#2i"
"IDP5.0.08.04, X604, TC#2i"
"IDP5.0.08.05, X605, TC#2i"
"IDP5.0.08.06, X606, TC#2i"
"IDP5.0.08.07, X607, TC#2i"
"IDP5.0.08.11, X611, TC#2i"
"IDP5.0.08.14, X614, TC#2i"
"IDP5.0.09.02, X702, TC#2i"
"IDP5.0.09.05, X705, TC#2i"
"IDP5.0.09.06, X706, TC#2i"
"IDP5.0.09.09, X709, TC#2i"
"IDP5.0.09.12, X712, TC#2i"
"IDP5.0.09.14, X714, TC#2i"
"IDP5.0.09.15, X715, TC#2i"
"IDP5.0.10.01, X801, TC#2i"
"IDP5.0.10.02, X802, TC#2i"
"IDP5.0.10.03, X803, TC#2i"
"IDP5.0.10.04, X804, TC#2i"
"IDP5.0.10.05, X805, TC#2i"
"IDP5.0.10.06, X806, TC#2i"
"IDP5.0.10.07, X807, TC#2i"
"IDP5.0.10.08, X808, TC#2i"
"IDP5.0.10.09, X809, TC#2i"
"IDP5.0.10.10, X810, TC#2i"
"IDP5.0.10.11, X811, TC#2i"
"IDP5.0.10.12, X812, TC#2i"
"IDP5.0.10.16, X816, TC#3i"
"QDP5.0.05.07, Y307, TC#2o"
"QDP5.0.05.14, Y314, TC#2o"
"QDP5.0.06.01, Y401, TC#2o"
"QDP5.0.06.02, Y402, TC#2o"
"QDP5.0.06.03, Y403, TC#2o"
"QDP5.0.06.04, Y404, TC#2o"
"QDP5.0.06.05, Y405, TC#2o"
"QDP5.0.06.06, Y406, TC#2o"
"QDP5.0.06.08, Y408, TC#2o"
"QDP5.0.06.09, Y409, TC#2o"
"QDP5.0.06.10, Y410, TC#2o"
"QDP5.0.06.12, Y412, TC#2o"
"QDP5.0.06.13, Y413, TC#2o"
"QDP5.0.06.14, Y414, TC#2o"
"QDP5.0.06.15, Y415, TC#2o"
"QDP5.0.07.01, Y501, TC#2o"
"QDP5.0.07.02, Y502, TC#2o"
"QDP5.0.07.03, Y503, TC#2o"
"QDP5.0.07.04, Y504, TC#2o"
"QDP5.0.07.05, Y505, TC#2o"
"QDP5.0.07.06, Y506, TC#2o"
"QDP5.0.07.07, Y507, TC#2o"
"QDP5.0.07.08, Y508, TC#2o"
"QDP5.0.07.09, Y509, TC#2o"
"QDP5.0.07.13, Y513, TC#2o"
"QDP5.0.08.04, Y604, TC#2o"
"QDP5.0.08.05, Y605, TC#2o"
"QDP5.0.08.06, Y606, TC#2o"
"QDP5.0.08.07, Y607, TC#2o"
"QDP5.0.08.08, Y608, TC#2o"
"QDP5.0.08.09, Y609, TC#2o"
"QDP5.0.09.14, Y714, TC#2o"
"QDP5.0.10.15, Y815, TC#3o"
"QDP5.0.10.16, Y816, TC#3o"
```

### Package Logical/Timestamp - Keeps current timestamp

### Timestamp.var - Global variables
```iecst
(********************************************************************
 * COPYRIGHT -- HP
 ********************************************************************
 * Package: Timestamp
 * File: Timestamp.var
 * Author: treamsbottom
 * Created: June 04, 2014
 ********************************************************************
 * Variables of package Timestamp
 ********************************************************************)
VAR
	CurrentTimestamp : DATE_AND_TIME;
END_VAR
```

### Package Logical/Data_BackUp - *Handles all data back up

### SQL.var - Global variables
```iecst
(********************************************************************
 * COPYRIGHT -- HP
 ********************************************************************
 * Package: SQL
 * File: SQL.var
 * Author: treamsbottom
 * Created: October 01, 2013
 ********************************************************************
 * Variables of package SQL
 ********************************************************************)
VAR
	SqlRequest : ARRAY[0..dec_c_MaxSQL] OF SQLRequest_typ;
	SQLBuffer : SQLRequest_typ;
END_VAR
VAR RETAIN
	SQL : SQL_Typ;
END_VAR
VAR
	Count : ARRAY[0..99] OF UDINT;
END_VAR
```

### Program Logical/SQL/zzSQLDriver (IEC) - *Driver to Handle SQL Requests

#### zzSQLDriver.var
```iecst
(********************************************************************
 * COPYRIGHT -- HP
 ********************************************************************
 * Program: zzSQLDriver
 * File: zzSQLDriver.var
 * Author: treamsbottom
 * Created: October 01, 2013
 ********************************************************************
 * Local variables of program zzSQLDriver
 ********************************************************************)
VAR
	LoginReq : BOOL;
	LoginTimer : BOOL;
	LoginTimerET : UDINT;
	x : UINT;
	SqlRequestLogin : BOOL;
	WriteToSql : SQL_Write;
	StringBuilt : BOOL;
	SqlCommandString : STRING[200];
END_VAR
VAR CONSTANT
	MaxBuffer : USINT := 10;
END_VAR
VAR
	ReadWriteSql : SQL_Read_Write;
	n : UINT;
	StartPosition : UINT;
END_VAR
```

#### zzSQLDriver.ab
```automation-basic
(********************************************************************
 * COPYRIGHT -- HP
 ********************************************************************
 * Program: zzSQLDriver
 * File: zzSQLDriver.ab
 * Author: treamsbottom
 * Created: October 01, 2013
 ********************************************************************
 * Implementation of program zzSQLDriver
 ********************************************************************)

PROGRAM _INIT

END_PROGRAM

PROGRAM _CYCLIC
//Allow PLC time to connect to SQL database or will continually request Log on Info
SqlRequestLogin = (D32[570] > 0) AND (D32[570] < 5);
TON_10ms((LoginReq AND NOT SqlRequestLogin),600,LoginTimer,LoginTimerET)
IF LoginTimer THEN
	D32[570] = 101
ENDIF

;Put all requests to SQL into the que Assign a ID so we know where to reply...
LOOP n = 0 TO dec_c_MaxSQL DO
	IF n >= StartPosition THEN
		IF SqlRequest[n].Request THEN ;New Request Not in Que
			IF (SQLBuffer.RequestID = 0) AND (SQLBuffer.RequestID = 0) THEN
				;Give New Sql Request ID
				SqlRequest[n].RequestID = n
				SQLBuffer = SqlRequest[n]
				StartPosition = n + 1
			ENDIF
		ENDIF
	ENDIF
	IF (SQLBuffer.RequestID = 0) AND (n >= dec_c_MaxSQL) THEN
		StartPosition = 0
	ENDIF
	EXITIF (SQLBuffer.RequestID > 0)
ENDLOOP
;SQL commands..
IF (SQLBuffer.RequestID > 0) THEN
	CASE SQLBuffer.SQLType OF

		ACTION cSQLType_WriteOnly:
			;Build SQL Request
			;IF NOT StringBuilt THEN
			strcpy(ADR(SqlCommandString),"")
			strcpy(ADR(SqlCommandString),ADR(cSqluspCommands[SQLBuffer.SQL_usp]))
			strcat(ADR(SqlCommandString),ADR(cSQL_Space))
			LOOP n = 0 TO SQLBuffer.NoOfParams - 1 DO
				strcat(ADR(SqlCommandString),ADR(SQLBuffer.Parameters[n].Param_String))
				IF n <> SQLBuffer.NoOfParams - 1 THEN
					strcat(ADR(SqlCommandString),ADR(cSQL_Comma_Space))
				ENDIF
				;No Output Strings allowed
			ENDLOOP
			StringBuilt = TRUE
			;ENDIF

			;Write Request
			WriteToSql.enable = StringBuilt
			WriteToSql.pDatabaseName = ADR(SQL.Login.DBName)
			WriteToSql.pServerName = ADR(SQL.Login.Path)
			WriteToSql.pUserName = ADR(SQL.Login.User)
			WriteToSql.pPassword = ADR(SQL.Login.Password)
			WriteToSql.pSQl_Cmd_String = ADR(SqlCommandString)
			WriteToSql FUB SQL_Write()
			IF WriteToSql.status = ERR_OK THEN
				;Write Complete Reset Request
				SqlRequest[SQLBuffer.RequestID].Complete = TRUE
				SQLBuffer = cEmptySQlReq
				StringBuilt = FALSE
				strcpy(ADR(SqlCommandString),"")
			ELSE IF WriteToSql.status <> ERR_FUB_BUSY THEN ; Error
				SqlRequest[SQLBuffer.RequestID].RequestID = 0
				SqlRequest[SQLBuffer.RequestID].Fail = TRUE
				SQLBuffer = cEmptySQlReq
			ENDIF
		ENDACTION

		ACTION cSQLType_ReadWrite:
			;Build SQL Request
			;IF NOT StringBuilt THEN
			strcpy(ADR(SqlCommandString),"")
			strcpy(ADR(SqlCommandString),ADR(cSqluspCommands[SQLBuffer.SQL_usp]))
			strcat(ADR(SqlCommandString),ADR(cSQL_Space))
			LOOP n = 0 TO SQLBuffer.NoOfParams - 1 DO
				strcat(ADR(SqlCommandString),ADR(SQLBuffer.Parameters[n].Param_String))
				IF n <> SQLBuffer.NoOfParams - 1 THEN
					strcat(ADR(SqlCommandString),ADR(cSQL_Comma_Space))
				ENDIF
				;No Output Strings allowed
			ENDLOOP
			StringBuilt = TRUE
			;ENDIF

			;Write Request
			ReadWriteSql.enable = StringBuilt
			ReadWriteSql.pDatabaseName = ADR(SQL.Login.DBName)
			ReadWriteSql.pServerName = ADR(SQL.Login.Path)
			ReadWriteSql.pUserName = ADR(SQL.Login.User)
			ReadWriteSql.pPassword = ADR(SQL.Login.Password)
			ReadWriteSql.pSQl_Cmd_String = ADR(SqlCommandString)
			ReadWriteSql.pData = ADR(SQLBuffer.OutputData[0])
			ReadWriteSql FUB SQL_Read_Write()
			IF ReadWriteSql.status = ERR_OK THEN
				;Write Complete Reset Request
				memcpy(ADR(SqlRequest[SQLBuffer.RequestID].OutputData[0]),ADR(SQLBuffer.OutputData[0]),SIZEOF(SQLBuffer.OutputData))
				SqlRequest[SQLBuffer.RequestID].Complete = TRUE
				SQLBuffer = cEmptySQlReq
				StringBuilt = FALSE
				strcpy(ADR(SqlCommandString),"")
			ELSE IF ReadWriteSql.status <> ERR_FUB_BUSY THEN ; Error
				SqlRequest[SQLBuffer.RequestID].RequestID = 0
				SqlRequest[SQLBuffer.RequestID].Fail = TRUE
				SQLBuffer = cEmptySQlReq
			ENDIF
		ENDACTION

		ACTION cSQLType_ReadOnly:
			;Build SQL Request
			;IF NOT StringBuilt THEN
			strcpy(ADR(SqlCommandString),"")
			strcpy(ADR(SqlCommandString),ADR(cSqluspCommands[SQLBuffer.SQL_usp]))
			StringBuilt = TRUE

			;Write Request
			ReadWriteSql.enable = StringBuilt
			ReadWriteSql.pDatabaseName = ADR(SQL.Login.DBName)
			ReadWriteSql.pServerName = ADR(SQL.Login.Path)
			ReadWriteSql.pUserName = ADR(SQL.Login.User)
			ReadWriteSql.pPassword = ADR(SQL.Login.Password)
			ReadWriteSql.pSQl_Cmd_String = ADR(SqlCommandString)
			ReadWriteSql.pData = ADR(SQLBuffer.OutputData[0])
			ReadWriteSql FUB SQL_Read_Write()
			IF ReadWriteSql.status = ERR_OK THEN
				;Write Complete Reset Request
				memcpy(ADR(SqlRequest[SQLBuffer.RequestID].OutputData[0]),ADR(SQLBuffer.OutputData[0]),SIZEOF(SQLBuffer.OutputData))
				SqlRequest[SQLBuffer.RequestID].Complete = TRUE
				SQLBuffer = cEmptySQlReq
				StringBuilt = FALSE
				strcpy(ADR(SqlCommandString),"")
			ELSE IF ReadWriteSql.status <> ERR_FUB_BUSY THEN ; Error
				SqlRequest[SQLBuffer.RequestID].RequestID = 0
				SqlRequest[SQLBuffer.RequestID].Fail = TRUE
				SQLBuffer = cEmptySQlReq
			ENDIF
		ENDACTION
	ENDCASE
ENDIF

END_PROGRAM
```

### Program Logical/SQL/zzTvText (IEC) - Text From TrackView

#### zzTvText.ab - Implementation code
```automation-basic
(********************************************************************
 * COPYRIGHT -- HP
 ********************************************************************
 * Program: zzTviewText
 * File: zzTviewText.ab
 * Author: Dave
 * Created: January 30, 2013
 ********************************************************************
 * Implementation of program zzTviewText
 ********************************************************************)

PROGRAM _INIT

StartSQLServerRead = TRUE
myRequest = 1

END_PROGRAM

PROGRAM _CYCLIC

	;Requests from TrackView
	;-----------------------

	;Read SQL Server connection values
	IF (NOT StartSQLServerRead AND (D32[570] = StartSQLServerDataRead)) THEN
		StartSQLServerRead 	= TRUE
		myRequest			= 1
	ENDIF

	IF StartSQLServerRead THEN

		IF myRequest = 1 THEN
			D32[220] = SendSUPDBServer
		ELSE IF myRequest = 2 THEN
			D32[220] = SendSUPDBName
		ELSE IF myRequest = 3 THEN
			D32[220] = SendSUPDBLogin
		ELSE IF myRequest = 4 THEN
			D32[220] = SendSUPDBPword
		ENDIF

		IF (D32[570] = D32[220]) THEN
			myRequest = myRequest + 1
		ENDIF

	ENDIF

	;Read all Textwords - example
	IF (NOT StartTextwords AND (D32[570] = StartReadTextwords)) THEN
		StartTextwords 		= TRUE
		myRequest			= 0
	ENDIF

	IF StartTextwords THEN

		D32[220] = (SendTextWord + myRequest)

		IF (D32[570] = D32[220]) THEN
			myRequest = myRequest + 1
		ENDIF

		IF (myRequest > 999) THEN
			StartTextwords 	= FALSE
			myRequest			= 0
			D32[220]			= 0
			D32[570] 			= 0
		ENDIF

	ENDIF

	;TrackView has sent some new Data - Replace / Add myTviewString with required variable
	IF (D32[570] > 0) AND (D32[570] = D32[220]) THEN
		IF D32[570] = SendSUPDBServer THEN
			memcpy(ADR(SQL.Login.Path),ADR(D32[571]),16)
			Login = RIGHT(SQL.Login.Path,5) ;Check if port number is set in trackview if not, Add port.
			result = strcmp(ADR(Login),ADR(SQL_Port))
			IF (result <> 0) THEN
				SQL.Login.Path =	CONCAT(SQL.Login.Path,SQL_Port)
			ENDIF
		ELSE IF D32[570] = SendSUPDBName THEN
			memcpy(ADR(SQL.Login.DBName),ADR(D32[571]),16)
		ELSE IF D32[570] = SendSUPDBLogin THEN
			memcpy(ADR(SQL.Login.User),ADR(D32[571]),16)
		ELSE IF D32[570] = SendSUPDBPword THEN
			memcpy(ADR(SQL.Login.Password),ADR(D32[571]),16)
		ELSE IF (D32[570] >= SendTextWord) AND (D32[570] <= SendTextWord + 999) THEN
			memcpy(ADR(myTviewString),ADR(D32[571]),16)
		ENDIF
	ENDIF
	IF StartSQLServerRead AND (myRequest > 4) THEN
		StartSQLServerRead 	= FALSE
		myRequest			= 0
		D32[220]			= 0
	ELSE IF StartTextwords AND (myRequest > 999) THEN
		StartTextwords 	= FALSE
		myRequest			= 0
		D32[220]			= 0
		D32[570] 			= 0
	ENDIF

END_PROGRAM
```

### Library Logical/SQL/zzSQL_Lib (IEC, version 1.00.1) - SQL_Function_Blocks
Depends on: AsDb, AsIecCon, AsTime, runtime, standard, AsString

#### zzSQL_Lib.fun - Exported functions and function blocks
```iecst
(********************************************************************
 * COPYRIGHT -- HP
 ********************************************************************
 * Library: zzSQL_Lib
 * File: zzSQL_Lib.fun
 * Author: treamsbottom
 * Created: May 04, 2012
 ********************************************************************
 * Functions and function blocks of library zzSQL_Lib
 ********************************************************************)

FUNCTION_BLOCK SQL_Write (**General Write to SWL Server. Set Data parameters in connection string.*)
	VAR_INPUT
		enable : BOOL;
		pServerName : UDINT;
		pUserName : UDINT;
		pPassword : UDINT;
		pDatabaseName : UDINT;
		pSQl_Cmd_String : UDINT;
	END_VAR
	VAR_OUTPUT
		status : UINT;
		sql_Error : UINT;
	END_VAR
	VAR
		SQL : SQL_Enum;
		internal_error : BOOL;
		SQLConnect : dbConnect;
		sql_Ident : UDINT;
		sql_Status : UINT;
		SQLExecute : dbExecuteSql;
		SQLDisconnect : dbDisconnect;
		SQLGetErrorMsg : dbGetErrorMessage;
		SQL_Error_Msg : STRING[100];
	END_VAR
END_FUNCTION_BLOCK

FUNCTION_BLOCK SQL_Read_Write (**SQL FB that return 20 UDINTS from Cat number*)
	VAR_INPUT
		pServerName : UDINT;
		pUserName : UDINT;
		pPassword : UDINT;
		pDatabaseName : UDINT;
		pData : UDINT;
		pSQl_Cmd_String : UDINT;
		enable : BOOL;
	END_VAR
	VAR_OUTPUT
		sql_Status : UINT;
		sql_Error : UINT;
		SQL_Error_Msg : STRING[100];
		status : UINT;
	END_VAR
	VAR
		SQL : SQL_Enum;
		Data : ARRAY[0..Dec_SqlOutputTypArrayLen] OF SQL_Output;
		sIndex : STRING[8];
		SQLConnect : dbConnect;
		sql_Ident : UDINT;
		SQLDisconnect : dbDisconnect;
		SQLExecute : dbExecuteSql;
		SQLFetchNextRow : dbFetchNextRow;
		n : UINT;
		SQLGetData : dbGetData;
		ColumnCount : UINT;
		SQlColumnCount : dbGetColumnCount;
		SQL_Data : BOOL;
		SQLGetErrorMsg : dbGetErrorMessage;
		internal_error : BOOL;
	END_VAR
END_FUNCTION_BLOCK
```

#### SQL_Write.ab - *General Write to SWL Server. Set Data parameters in connection string.
```automation-basic
(********************************************************************
 * COPYRIGHT -- HP
 ********************************************************************
 * Library: zzSQL_Lib
 * File: SQL_Write.ab
 * Author: treamsbottom
 * Created: May 10, 2012
 ********************************************************************
 * Implementation of library zzSQL_Lib
 ********************************************************************)

(* *General Write to SWL Server. Set Data parameters in connection string. *)
FUNCTION_BLOCK SQL_Write
status = ERR_FUB_BUSY

IF NOT enable AND (SQL <> eConnect)  THEN
	SQL = eDisconnect
ENDIF
CASE SQL OF

	ACTION eConnect:
		internal_error = FALSE
		SQLConnect.enable 			= enable ;AND NOT internal_error
		SQLConnect.pServerName 		= pServerName;ADR("10.0.10.1:1433")
		SQLConnect.pUserName		= pUserName;ADR("SUP")
		SQLConnect.pPassword		= pPassword;ADR("1234")
		SQLConnect.pDatabaseName	= pDatabaseName;ADR("SUPDB1")
		SQLConnect.databaseSystem 	= DB_SYSTEM_MS_SQL
		SQLConnect FUB dbConnect()

		sql_Ident = SQLConnect.connectionIdent
		sql_Status = SQLConnect.status
		sql_Error = SQLConnect.dbError
		IF sql_Status = ERR_OK THEN
			SQL = eExecute
			;SQL = eIdle
		ELSE IF sql_Status <> ERR_FUB_BUSY THEN
			status = sql_Status
			SQL = eError
		ENDIF
	ENDACTION

	ACTION eExecute:
		SQLExecute.enable 			= TRUE
		SQLExecute.connectionIdent 	= sql_Ident
		SQLExecute.pSqlStatement 	= pSQl_Cmd_String
		SQLExecute FUB dbExecuteSql()
		IF SQLExecute.status = ERR_OK THEN
			SQL = eDisconnect
			;SQL = eIdle
		ELSE IF SQLExecute.status <> ERR_FUB_BUSY THEN
			status = SQLExecute.status
			SQL = eError
			sql_Error = SQLExecute.dbError
			sql_Status = SQLExecute.status
		ENDIF
	ENDACTION

	ACTION eDisconnect:
		SQLDisconnect.enable 			= TRUE
		SQLDisconnect.connectionIdent 	= sql_Ident
		SQLDisconnect FUB dbDisconnect()
		sql_Status = SQLDisconnect.status
		IF SQLDisconnect.status = ERR_OK THEN
			;enable = FALSE
			IF internal_error THEN

			ELSE
				status = ERR_OK
			ENDIF
			SQL = eConnect
		ELSE IF SQLDisconnect.status = dbERR_INVALID_HANDLE THEN ; Ident not valid
			SQL = eConnect
		ENDIF
	ENDACTION

	ACTION eError:
		internal_error = TRUE
		SQLGetErrorMsg.enable = TRUE
		SQLGetErrorMsg.connectionIdent = sql_Ident
		SQLGetErrorMsg.pErrorMessage = ADR(SQL_Error_Msg)
		SQLGetErrorMsg.errorMessageSize = SIZEOF(SQL_Error_Msg)
		SQLGetErrorMsg FUB dbGetErrorMessage()
		IF SQLGetErrorMsg.status = ERR_OK THEN
			IF sql_Ident = 0 THEN
				SQL = eConnect
				;enable = FALSE
			ELSE
				SQL = eDisconnect
			ENDIF
		ELSE IF (SQLGetErrorMsg.status <> ERR_FUB_BUSY) THEN
			IF sql_Ident = 0 THEN
				SQL = eConnect
			ELSE
				SQL = eDisconnect
			ENDIF
		ENDIF
	ENDACTION

ENDCASE

END_FUNCTION_BLOCK
```

#### SQL_Read_Write.ab - *SQL FB that return 20 UDINTS from Cat number
```automation-basic
(********************************************************************
 * COPYRIGHT -- HP
 ********************************************************************
 * Library: zzSQL_Lib
 * File: SQL_D32.ab
 * Author: treamsbottom
 * Created: May 08, 2012
 ********************************************************************
 * Implementation of library zzSQL_Lib
 ********************************************************************)

(* *SQL FB that return 20 UDINTS from Cat number *)
FUNCTION_BLOCK SQL_Read_Write

SQL_Data = TRUE
status = ERR_FUB_BUSY

IF NOT enable AND (SQL <> eConnect)  THEN
	SQL = eDisconnect
ENDIF
CASE SQL OF

	ACTION eConnect:
		internal_error = FALSE
		SQLConnect.enable 			= enable ;AND NOT internal_error
		SQLConnect.pServerName 		= pServerName;ADR("10.0.10.1:1433")
		SQLConnect.pUserName		= pUserName;ADR("SUP")
		SQLConnect.pPassword		= pPassword;ADR("1234")
		SQLConnect.pDatabaseName	= pDatabaseName;ADR("SUPDB1")
		SQLConnect.databaseSystem 	= DB_SYSTEM_MS_SQL
		SQLConnect FUB dbConnect()

		sql_Ident = SQLConnect.connectionIdent
		sql_Status = SQLConnect.status
		sql_Error = SQLConnect.dbError
		IF sql_Status = ERR_OK THEN
			SQL = eExecute
			;SQL = eIdle
		ELSE IF sql_Status <> ERR_FUB_BUSY THEN
			status = sql_Status
			SQL = eError
		ENDIF
	ENDACTION

	ACTION eExecute:
		SQLExecute.enable 			= TRUE
		SQLExecute.connectionIdent 	= sql_Ident
		SQLExecute.pSqlStatement 	= pSQl_Cmd_String
		SQLExecute FUB dbExecuteSql()
		IF SQLExecute.status = ERR_OK THEN
			SQL = eReadData
			;SQL = eIdle
		ELSE IF SQLExecute.status <> ERR_FUB_BUSY THEN
			status = SQLExecute.status
			SQL = eError
			sql_Error = SQLExecute.dbError
			sql_Status = SQLExecute.status
		ENDIF
	ENDACTION

	ACTION eReadData:
		SQLFetchNextRow.enable = TRUE
		SQLFetchNextRow.connectionIdent = sql_Ident
		SQLFetchNextRow FUB dbFetchNextRow()
		IF SQLFetchNextRow.status = ERR_OK THEN
			n = 1
			SQL = eColumnCount
			;SQL = eIdle
		ELSE IF SQLFetchNextRow.status = dbERR_DATABASE THEN; No valid data
			status = SQLFetchNextRow.status
			SQL = eDisconnect
			SQL_Data = FALSE
		ELSE IF	SQLFetchNextRow.status <> ERR_FUB_BUSY THEN
			status = SQLFetchNextRow.status
			sql_Error 	=  SQLFetchNextRow.dbError
			sql_Status 	= SQLFetchNextRow.status
			SQL = eError
		ENDIF
	ENDACTION

	ACTION eColumnCount:
		SQlColumnCount.enable 			= TRUE
		SQlColumnCount.connectionIdent 	= sql_Ident
		SQlColumnCount FUB dbGetColumnCount()
		IF SQlColumnCount.status = ERR_OK THEN
			ColumnCount = SQlColumnCount.columnCount
			;SQL = eIdle
			IF ColumnCount > 0 THEN
				SQL = eGetData
				SQL_Data = TRUE
				n = 1
			ELSE
				SQL = eDisconnect
				SQL_Data = FALSE
			ENDIF
		ELSE IF SQlColumnCount.status <> ERR_FUB_BUSY THEN
			status = SQlColumnCount.status
			SQL = eError
		ENDIF
	ENDACTION

	ACTION eGetData:

		SQLGetData.enable 			= TRUE
		SQLGetData.connectionIdent	= sql_Ident
		SQLGetData.columnIdx		= n ; Columns Start from 1, 0 will return an error
		SQLGetData.dataType			= DB_SQL_CHAR ; Variable String
		SQLGetData.pData			= ADR(Data[n])
		SQLGetData.dataSize			= SIZEOF(Data[n])
		SQLGetData	FUB dbGetData()
		IF SQLGetData.status = ERR_OK THEN

			IF n = ColumnCount THEN
				;Cope Data to Out variable
				memcpy(pData,ADR(Data),SIZEOF(Data))
				SQL = eDisconnect
			ENDIF
			n = n + 1
		ELSE IF SQLGetData.status <> ERR_FUB_BUSY THEN
			status = SQLGetData.status
			sql_Error 	=  SQLGetData.dbError
			sql_Status 	= SQLGetData.status
			SQL = eError
		ENDIF
	ENDACTION

	ACTION eDisconnect:
		SQLDisconnect.enable 			= TRUE
		SQLDisconnect.connectionIdent 	= sql_Ident
		SQLDisconnect FUB dbDisconnect()
		sql_Status = SQLDisconnect.status
		IF SQLDisconnect.status = ERR_OK THEN
			;enable = FALSE
			IF internal_error THEN
				status = 20
			ELSE
				status = ERR_OK
			ENDIF
			;SQL = eConnect
		ELSE IF SQLDisconnect.status = dbERR_INVALID_HANDLE THEN ; Ident not valid
			SQL = eConnect
		ENDIF
	ENDACTION

	ACTION eError:
		internal_error = TRUE
		SQLGetErrorMsg.enable = TRUE
		SQLGetErrorMsg.connectionIdent = sql_Ident
		SQLGetErrorMsg.pErrorMessage = ADR(SQL_Error_Msg)
		SQLGetErrorMsg.errorMessageSize = SIZEOF(SQL_Error_Msg)
		SQLGetErrorMsg FUB dbGetErrorMessage()
		IF SQLGetErrorMsg.status = ERR_OK THEN
			IF sql_Ident = 0 THEN
				SQL = eConnect
				;enable = FALSE
			ELSE
				SQL = eDisconnect
			ENDIF
		ELSE IF (SQLGetErrorMsg.status <> ERR_FUB_BUSY) THEN
			IF sql_Ident = 0 THEN
				SQL = eConnect
			ELSE
				SQL = eDisconnect
			ENDIF
		ENDIF
	ENDACTION

ENDCASE

END_FUNCTION_BLOCK
```

### Program Logical/SQL/SQLReadWriteTest (IEC) - Program

#### SQLSpeedTest.var
```iecst
(********************************************************************
 * COPYRIGHT -- HP
 ********************************************************************
 * Program: SQLSpeedTest
 * File: SQLSpeedTest.var
 * Author: treamsbottom
 * Created: October 03, 2013
 ********************************************************************
 * Local variables of program SQLSpeedTest
 ********************************************************************)
VAR
	Sql : INT;
	SqlConnect : dbConnect;
	Ident : UDINT;
	SqlDisconnect : dbDisconnect;
	ConnectionCount : UINT;
	pServer : UDINT;
	pDatabaseName : UDINT;
	pUserName : UDINT;
	pPassword : UDINT;
	SqlError : dbGetErrorMessage;
	ErrorString : STRING[100];
	SqlExecute : dbExecuteSql;
	pServerName : UDINT;
	Break : UDINT;
	TestVar : UDINT;
	SqlColumnCount : dbGetColumnCount;
	ColumnCount : UDINT;
	SqlGetData : dbGetData;
	OutputDataRow : ARRAY[0..19] OF STRING[25];
	Row : INT;
	Col : INT;
	ReadData : USINT;
	SqlGetRow : dbFetchNextRow;
END_VAR
```

#### SQLSpeedTestCyclic.ab
```automation-basic
(********************************************************************
 * COPYRIGHT -- HP
 ********************************************************************
 * Program: SQLSpeedTest
 * File: SQLSpeedTestCyclic.ab
 * Author: treamsbottom
 * Created: October 03, 2013
 ********************************************************************
 * Implementation of program SQLSpeedTest
 ********************************************************************)
PROGRAM _INIT
Sql = 0

END_PROGRAM
PROGRAM _CYCLIC

pServer = ADR("10.8.4.210:1433")
pDatabaseName = ADR("SUPDB1")
pUserName = ADR("SUP")
pPassword = ADR("1234")
;	IF pServer <> TestVar THEN
;		INC Break
;		strcpy(ADR(ErrorString),pServer)
;	ENDIF

CASE Sql OF

	ACTION 50:
		SqlConnect.enable = TRUE
		SqlConnect.pServerName = ADR("10.8.4.210:1433")
		SqlConnect.pDatabaseName = ADR("SUPDB1")
		SqlConnect.pUserName = ADR("SUP")
		SqlConnect.pPassword = ADR("1234")
		SqlConnect.databaseSystem = DB_SYSTEM_MS_SQL
		SqlConnect FUB dbConnect()

		IF SqlConnect.status = ERR_OK THEN

			Ident = SqlConnect.connectionIdent
			IF Ident > 0 THEN
				Sql = 1
				INC ConnectionCount
			ENDIF
		ELSE IF SqlConnect.status <> ERR_FUB_BUSY THEN
			IF SqlConnect.connectionIdent <> 0 THEN
				Ident = SqlConnect.connectionIdent
				Sql = 99
			ENDIF
		ELSE IF Ident <> 0 THEN; Connection already made disconnect
			Sql = 2
		ENDIF
	ENDACTION

	ACTION 1:
		SqlExecute.enable = TRUE
		SqlExecute.connectionIdent = Ident
		SqlExecute.pSqlStatement = ADR("EXEC Supertrack.uspBagMaintCountReplyState 2 ,PLCReadWriteTest")
		SqlExecute FUB dbExecuteSql()
		IF SqlExecute.status = ERR_OK THEN
			ReadData = 1
			Sql = 2
		ENDIF
	ENDACTION

	ACTION 2:
		CASE ReadData OF
			ACTION 1: ; Fetch Data
				SqlGetRow.enable = TRUE
				SqlGetRow.connectionIdent = Ident
				SqlGetRow FUB dbFetchNextRow()
				IF SqlGetRow.status = ERR_OK THEN
					ReadData = 2
				ENDIF
			ENDACTION

			ACTION 2: ; Get results
				SqlColumnCount.enable = TRUE
				SqlColumnCount.connectionIdent = Ident
				SqlColumnCount FUB dbGetColumnCount()
				IF SqlColumnCount.status = ERR_OK THEN
					ColumnCount = SqlColumnCount.columnCount
					Col = 1
					Row = 0
					ReadData = 3
				ENDIF
			ENDACTION

			ACTION 3:
				SqlGetData.enable = TRUE
				SqlGetData.connectionIdent = Ident
				SqlGetData.dataType = DB_SQL_INTEGER ; Always read out as string
				SqlGetData.dataSize = SIZEOF(OutputDataRow[Row].Data[Col])
				SqlGetData.pData = ADR(OutputDataRow[Row].Data[Col])
				SqlGetData.columnIdx = Col
				SqlGetData FUB dbGetData()
				IF SqlGetData.status = ERR_OK THEN
;					IF Col = ColumnCount THEN
;						Col = 1
;						ReadData = 0
;						INC Row
;					ELSE
;						INC Col
;					ENDIF
					Sql = 78
				ENDIF
			ENDACTION
		ENDCASE
	ENDACTION

	ACTION 10:
		SqlDisconnect.enable = TRUE
		SqlDisconnect.connectionIdent = Ident
		SqlDisconnect FUB dbDisconnect()
		IF SqlDisconnect.status =  ERR_OK THEN
			Ident = 0
			Sql = 85
		ENDIF
	ENDACTION

	ACTION 99:
		SqlError.enable = TRUE
		SqlError.connectionIdent = Ident
		SqlError.pErrorMessage = ADR(ErrorString)
		SqlError.errorMessageSize = SIZEOF(ErrorString)
		SqlError FUB dbGetErrorMessage()
		IF SqlError.status = ERR_OK THEN
			Sql = 10
		ENDIF
	ENDACTION
ENDCASE

END_PROGRAM
```

### Program Logical/SQL/SQLSpeedTest (IEC) - Program

#### SQLSpeedTest.var - Local variables
```iecst
(********************************************************************
 * COPYRIGHT -- HP
 ********************************************************************
 * Program: SQLSpeedTest
 * File: SQLSpeedTest.var
 * Author: treamsbottom
 * Created: October 03, 2013
 ********************************************************************
 * Local variables of program SQLSpeedTest
 ********************************************************************)
VAR
	Sql : INT;
	SqlConnect : dbConnect;
	Ident : UDINT;
	SqlDisconnect : dbDisconnect;
	ConnectionCount : UINT;
	pServer : UDINT;
	pDatabaseName : UDINT;
	pUserName : UDINT;
	pPassword : UDINT;
	SqlError : dbGetErrorMessage;
	ErrorString : STRING[100];
	SqlExecute : dbExecuteSql;
	pServerName : UDINT;
	Break : UDINT;
	TestVar : UDINT;
END_VAR
```


- Program Logical/SQL/zzGetNamesSQL/zzGetNameSQL (IEC) - Get Names for Display (no source held here)

### Program Logical/SQL/Test_bagMaint (IEC) - Program

#### Test_bagMaint.ab - Implementation code
```automation-basic
(********************************************************************
 * COPYRIGHT -- HP
 ********************************************************************
 * Program: Test_bagMaint
 * File: Test_bagMaint.ab
 * Author: treamsbottom
 * Created: May 05, 2015
 ********************************************************************
 * Implementation of program Test_bagMaint
 ********************************************************************)

PROGRAM _INIT

(* TODO : Add your code here *)

END_PROGRAM

PROGRAM _CYCLIC

	strcpy(ADR(myBagNumber),"1")
	mySql = 88

	CASE TEST_STATE OF
		ACTION 0:

		ENDACTION

		ACTION 1: ; TEST WRITE COUNT
			SqlRequest[mySql].Request = TRUE
			IF SqlRequest[mySql].Complete THEN
				TEST_STATE = 0

			ENDIF
			IF SqlRequest[mySql].Request AND NOT SqlWriteActive THEN ; Write Count to SQL
				SqlWriteActive = TRUE
				SqlRequest[mySql].SQLType = cSQLType_WriteOnly
				SqlRequest[mySql].SQL_usp = cSQLReq_BagMaintCount
				SqlRequest[mySql].NoOfParams = 2

				SqlRequest[mySql].Parameters[0].Type = cSQLParam_Input ;PLC Stn
				strcpy(ADR(SqlRequest[mySql].Parameters[0].Param_String),ADR(Std.PLCStnString))
				SqlRequest[mySql].Parameters[1].Type = cSQLParam_Input ;BatchID;
				strcpy(ADR(SqlRequest[mySql].Parameters[1].Param_String),ADR(myBagNumber))
			ENDIF
		ENDACTION

		ACTION 2: ; TEST READ State
			SqlRequest[mySql].Request = TRUE
			IF SqlRequest[mySql].Complete THEN
				myBagState = UINT(atoi(ADR(SqlRequest[mySql].OutputData[1])))
				TEST_STATE = 0
			ELSE
				myBagState = 99
			ENDIF
			IF SqlRequest[mySql].Request AND NOT SqlWriteActive THEN ; Write Count to SQL
				SqlWriteActive = TRUE
				SqlRequest[mySql].SQLType = cSQLType_ReadWrite
				SqlRequest[mySql].SQL_usp = cSQLReq_BagMaintGetState
				SqlRequest[mySql].NoOfParams = 2

				SqlRequest[mySql].Parameters[0].Type = cSQLParam_Input ;PLC Stn
				strcpy(ADR(SqlRequest[mySql].Parameters[0].Param_String),ADR(Std.PLCStnString))
				SqlRequest[mySql].Parameters[1].Type = cSQLParam_Input ;BatchID;
				strcpy(ADR(SqlRequest[mySql].Parameters[1].Param_String),ADR(myBagNumber))
			ENDIF
		ENDACTION

		ACTION 3: ; TEST READ State
			SqlRequest[mySql].Request = TRUE
			IF SqlRequest[mySql].Complete THEN
				myBagState = UINT(atoi(ADR(SqlRequest[mySql].OutputData[1])))
				TEST_STATE = 0
			ELSE
				myBagState = 99
			ENDIF
			IF SqlRequest[mySql].Request AND NOT SqlWriteActive THEN ; Write Count to SQL
				SqlWriteActive = TRUE
				SqlRequest[mySql].SQLType = cSQLType_ReadWrite
				SqlRequest[mySql].SQL_usp = cSQLReq_BagMaintCount_R_State
				SqlRequest[mySql].NoOfParams = 2

				SqlRequest[mySql].Parameters[0].Type = cSQLParam_Input ;PLC Stn
				strcpy(ADR(SqlRequest[mySql].Parameters[0].Param_String),ADR(Std.PLCStnString))
				SqlRequest[mySql].Parameters[1].Type = cSQLParam_Input ;BatchID;
				strcpy(ADR(SqlRequest[mySql].Parameters[1].Param_String),ADR(myBagNumber))
			ENDIF
		ENDACTION

	ENDCASE

;**********************************************************************************
; Normally Code sits at bottom of task and we only pass SqlRequest[mySql].Request
;************************************************************************************

;IF SqlRequest[mySql].Request AND NOT SqlWriteActive THEN ; Write Count to SQL
;	SqlWriteActive = TRUE
;	SqlRequest[mySql].SQLType = cSQLType_ReadWrite
;	SqlRequest[mySql].SQL_usp = cSQLReq_BagMaintCount
;	SqlRequest[mySql].NoOfParams = 3
;
;	SqlRequest[mySql].Parameters[0].Type = cSQLParam_Input ;PLC Stn
;	strcpy(ADR(SqlRequest[mySql].Parameters[0].Param_String),ADR(Std.PLCStnString))
;	SqlRequest[mySql].Parameters[1].Type = cSQLParam_Input ;BatchID;
;	strcpy(ADR(SqlRequest[mySql].Parameters[1].Param_String),ADR(myBagNumber))
;ENDIF

IF SqlRequest[mySql].Complete THEN ; ClearRequest
	;Copy Out Reply Done in step.!
	SqlRequest[mySql] = cEmptySQlReq
	SqlWriteActive = FALSE
ELSE IF SqlRequest[mySql].Fail THEN
	WaitReply = FALSE ; Move to next and try and again
	SqlWriteActive = FALSE ; Reload Parameters
	SqlRequest[mySql].Fail = FALSE
ENDIF

END_PROGRAM
```

### Global.typ
```iecst
TYPE
	Alm : 	STRUCT
		On : BOOL;
		Bag : UINT;
		ET : TIME;
		InList : BOOL;
		Name : UINT;
		Extra : UINT;
		Beacon : BOOL;
		Time : UDINT;
	END_STRUCT;
	BagType : 	STRUCT
		Cat : USINT;
		Dst : USINT;
		Wgt : UINT;
		Cnt : UINT;
		Cus : UINT;
		Day : USINT;
		Spare : USINT;
	END_STRUCT;
	CardInputs : 	STRUCT
		X01 : BOOL;
		X02 : BOOL;
		X03 : BOOL;
		X04 : BOOL;
		X05 : BOOL;
		X06 : BOOL;
		X07 : BOOL;
		X08 : BOOL;
		X09 : BOOL;
		X10 : BOOL;
		X11 : BOOL;
		X12 : BOOL;
		X13 : BOOL;
		X14 : BOOL;
		X15 : BOOL;
		X16 : BOOL;
	END_STRUCT;
	CardOutputs : 	STRUCT
		Y01 : BOOL;
		Y02 : BOOL;
		Y03 : BOOL;
		Y04 : BOOL;
		Y05 : BOOL;
		Y06 : BOOL;
		Y07 : BOOL;
		Y08 : BOOL;
		Y09 : BOOL;
		Y10 : BOOL;
		Y11 : BOOL;
		Y12 : BOOL;
		Y13 : BOOL;
		Y14 : BOOL;
		Y15 : BOOL;
		Y16 : BOOL;
	END_STRUCT;
	DAM : 	STRUCT
		Alive : UINT;
		Analog : INT;
	END_STRUCT;
	Enable_Vars : 	STRUCT
		Search : UINT;
		TransferBelt : BOOL;
		Ongoing : ARRAY[0..4]OF BOOL;
		Offgoing : ARRAY[0..4]OF BOOL;
		SBS : ARRAY[0..4]OF BOOL;
		CLU : ARRAY[0..9]OF BOOL;
		CIC : ARRAY[0..9]OF BOOL;
		CDC : ARRAY[0..9]OF BOOL;
		CP : ARRAY[0..9]OF BOOL;
		SPN : ARRAY[0..9]OF BOOL;
		SVC : ARRAY[0..9]OF BOOL;
		SWB : ARRAY[0..4]OF BOOL;
		SPF : ARRAY[0..1]OF BOOL;
		CDC4Empty : BOOL;
		CDC4Open : BOOL;
		CVC : ARRAY[0..3]OF BOOL;
	END_STRUCT;
	Line_Vars : 	STRUCT
		Clear : BOOL;
		Full : BOOL;
		Trip : BOOL;
		FirstBag : UINT;
		LastBag : UINT;
		Space : UINT;
		SpaceBIT : UINT;
	END_STRUCT;
	Loading_Vars : 	STRUCT
		StartStn : UINT;
		EndStn : UINT;
		EnableStnRelease : BOOL;
		BeltHasRun : BOOL;
		Found : UINT;
		Line : UINT;
		Search : UINT;
	END_STRUCT;
	ReadDisplay : 	STRUCT
		Data : ARRAY[0..7]OF USINT;
	END_STRUCT;
	Reports : 	STRUCT
		Cat : UINT;
		Cus : UINT;
		Wgt : UINT;
		Cnt : UINT;
		Stn : UINT;
		Mcn : UINT;
	END_STRUCT;
	Request_Vars : 	STRUCT
		SDC1 : BOOL;
		SDC2 : BOOL;
		SDC2Full : BOOL;
		SIC1 : BOOL;
		SPF : BOOL;
		SVC1 : BOOL;
		TransferBelt : BOOL;
	END_STRUCT;
	ScanTime : 	STRUCT
		Start : TIME;
		End : TIME;
		Time : UINT;
		Min : UINT;
		Max : UINT;
	END_STRUCT;
	Std_Vars : 	STRUCT
		HaltSys : BOOL;
		HaltSysLoading : BOOL;
		StopSystem : BOOL;
		SafetyOn : BOOL;
		SafetyOnLoading : BOOL;
		AutoMaticRelease : BOOL;
		AutoRecirculation : BOOL;
		BagsWithDestinations : BOOL;
		BagsWithDestinations2 : BOOL;
		BagWithDestAtFront : BOOL;
		BagSpacing : USINT;
		Clock100ms : BOOL;
		Clock200ms : BOOL;
		Clock500ms : BOOL;
		Clock1s : BOOL;
		Clock2s : BOOL;
		EStop : BOOL;
		EStopLoading : BOOL;
		EnableOverUnderRelease : BOOL;
		MaxCats : USINT;
		MaxCust : UINT;
		MaxDischargers : USINT;
		MaxIO : UINT;
		MaxLines : UINT;
		MaxLinesBuffers : UINT;
		MaxWeighstations : UINT;
		MaxCountingStations : UINT;
		MaxStationBanks : UINT;
		MaxSearch : UINT;
		MinReleaseWeight : UINT;
		Monitor : UINT;
		MotorOverload : BOOL;
		MotorOverloadLoading : BOOL;
		PairingLoop : BOOL;
		Purging : BOOL;
		PurgeCompleted : BOOL;
		RepSpacing : USINT;
		StnBatchCode : UINT;
		StnsInQ : BOOL;
		StnsToPurge : BOOL;
		StationBagsStart : ARRAY[0..4]OF UINT;
		CountingBagsStart : UINT;
		StationReports : BOOL;
		StationsClosed : BOOL;
		TransferBeltRun : BOOL;
		UnloadingMaxDepth : UINT;
		CustomerFIFO : BOOL;
		CustomerFound : BOOL;
		AutoLineAllocation : BOOL;
		CustomerNewFound : BOOL;
		CustomerEditFound : BOOL;
	END_STRUCT;
	Stn_Mix : 	STRUCT
		Cat : ARRAY[0..9]OF UINT;
		Cus : ARRAY[0..9]OF UINT;
		Wgt : ARRAY[0..9]OF UINT;
		Cnt : ARRAY[0..9]OF UINT;
	END_STRUCT;
	Stn_Vars : 	STRUCT
		DestManual : UINT;
		LampOn : BOOL;
		ManualRelease : BOOL;
		QTime : UINT;
		ReleaseButton : BOOL;
		SpacesRequired : UINT;
		SP1 : BOOL;
		SP2 : BOOL;
		SP3 : BOOL;
		Count : UINT;
		Reg : UINT;
		Closed : BOOL;
		CntInput : BOOL;
		Weight : INT;
		Open : BOOL;
		PBCount : UINT;
		LampFlashFast : BOOL;
		CloseFlap : BOOL;
		Unlock : BOOL;
	END_STRUCT;
	Test_Vars : 	STRUCT
		TransferBelt : BOOL;
		Stations : BOOL;
		Dropped : ARRAY[0..4]OF BOOL;
		Drop : ARRAY[0..4]OF BOOL;
		Dischargers : BOOL;
	END_STRUCT;
	Uld_Vars : 	STRUCT
		SDCReady : BOOL;
		SDCSpaces : UINT;
		DischargerStartLine : UINT;
		LastCustQtyComplete : UINT;
		FIFOCustomer : UINT;
		FIFOCustomerFound : BOOL;
		FIFONextCustomer : UINT;
	END_STRUCT;
	WriteDisplay : 	STRUCT
		Data : ARRAY[0..7]OF USINT;
	END_STRUCT;
	comstype : 	STRUCT
		delime : UINT;
		delim : ARRAY[0..1]OF USINT;
		tx_cnt : UINT;
		rx_cnt : UINT;
		tx_len : UINT;
		rx_len : UINT;
		argc : UINT;
		argv : UDINT;
		idle : UINT;
	END_STRUCT;
	fiLOCAL_OBJ : 	STRUCT
		StateMan : UINT;
		ErrMan : UINT;
		Init : UDINT;
	END_STRUCT;
END_TYPE
```

### Global.var
```iecst
VAR RETAIN
	Alarm : ARRAY[0..109] OF Alm;
	AlarmBagNotProxLine : UINT;
	Bag : ARRAY[0..999] OF BagType;
	C : ARRAY[0..99] OF UINT;
	D : ARRAY[0..5999] OF UINT;
	Enable : Enable_Vars;
	Ldg : ARRAY[0..4] OF Loading_Vars;
	Line : ARRAY[0..99] OF Line_Vars;
	ReportBuffer : ARRAY[0..199] OF Reports;
	ReportLoading : ARRAY[0..50] OF Reports;
	ReportUnloading : ARRAY[0..10] OF Reports;
	Request : Enable_Vars;
	Std : Std_Vars;
	Stn : ARRAY[0..50] OF Stn_Vars;
	TCScan : ARRAY[0..8] OF ScanTime;
	Test : Test_Vars;
	Uld : ARRAY[0..20] OF Uld_Vars;
END_VAR
VAR CONSTANT
	almBagDataError : UINT := 20;
	almBagNotArrived : UINT := 6;
	almBagNotAtProx : UINT := 16;
	almBagNotReleased : UINT := 9;
	almBagNotSettled : UINT := 7;
	almEmergencyStop : UINT := 1;
	almGeneralSequence : UINT := 15;
	almInverterFault : UINT := 18;
	almLoadNotDropped : UINT := 10;
	almMotorOverload : UINT := 2;
	almNoAlarm : UINT := 0;
	almSwitchFault : UINT := 5;
	almUldNoBag : UINT := 4;
	almUldProgFinished : UINT := 3;
END_VAR
VAR
	AI354RAW_1 : INT; (* ±10 V, resolution 12 bit *)
	AI354RAW_2 : INT; (* ±10 V, resolution 12 bit *)
	AI354RAW_3 : INT; (* ±10 V, resolution 12 bit *)
	AI354RAW_4 : INT; (* ±10 V, resolution 12 bit *)
	I_EStop : BOOL;
	Indication : ARRAY[0..79] OF BOOL;
	SSS2Raw : DINT;
	SSS2Weight : UINT;
	SSS3Raw : DINT;
	SSS3Weight : UINT;
	SSS4Raw : DINT;
	SSS4Weight : UINT;
	StnPrev : ARRAY[0..50] OF BagType;
	TimerAlarm : TON_10ms;
	X : ARRAY[0..39] OF CardInputs;
	Y : ARRAY[0..39] OF CardOutputs;
	YForceDisable : ARRAY[0..39] OF CardOutputs;
	Zero : UINT := 0;
	pBag : UDINT;
	pC : UDINT;
	pD : UDINT;
END_VAR
```

- Program Logical/zzclrmem (IEC, version 2.00.0) - * Clear Permanent Memory (no source held here)

### Program Logical/zzweigh (IEC, version 3.00.0) - * Station Weight Calculation and Calibration

#### zzweighCyclic.ab
```automation-basic
PROGRAM _CYCLIC
	(* cyclic program *)

;---------------------------------------------------------------------------------------------
;Revision 1.00 01/05/2001 D.J. First Issue
;Revision 2.00 23/10/2002 D.J. WeightUnits changed to DINT (problem when raw values over 32767
;Revision 3.00 22/08/2006 D.J. Changed for AI261
;---------------------------------------------------------------------------------------------

;------------------------------------------------------------
;WeighStation Calibration and Weight Calculation - With AI261
;------------------------------------------------------------

;divide by 1000 should give around 50 parts per kg and keep raw value within UINT
;Add 32000 to value to ensure always positive
LOOP n = 1 TO Std.MaxWeighstations DO
	;To view a particular stn then set tstRaw to the required stn
	IF tstRaw > 0 THEN
		myRaw = tstRaw ;AI261Raw[tstRaw]
	ELSE
	;	myRaw = AI2744Raw[n]????????????????????????????????????????????????
	ENDIF
	;Ensure raw value is within + 24bit if out of range + 32bit
	IF (myRaw = $7FFFFFFF) THEN
		myRaw = $FFFFFF
	ENDIF
	;Ensure raw value is within - 24bit if out of range - 32bit
	IF (myRaw = $80000001) THEN
		myRaw = $FF000001
	ENDIF
	;Convert raw to UINT the 3 least significant digits are removed
	myStnRaw = UINT((myRaw / 1000) + 32000)
	StnRaw[n] = myStnRaw
ENDLOOP

LOOP n = 1 TO Std.MaxWeighstations DO

	StnLow 		= D[3400 + n]
	StnHigh 	= D[3500 + n]
	StnTestWgt 	= D[3600 + n]

	;Calibrate Low - From TrackView
	IF (D[995] = n) AND (D[996] = 11) THEN
		NewLow = StnRaw[n]
		IF (NewLow > 0) AND (NewLow < $FFFF) THEN
			D[3400 + n] = NewLow
		ENDIF
		D[996] = 0 ;Cancel the Cal-Low
	ENDIF
	;Calibrate High - From TrackView
	IF (D[995] = n) AND (D[996] = 12) AND (D[997] > 0) THEN
		NewHigh = StnRaw[n]
		IF (NewHigh > 0) AND (NewHigh < $FFFF) AND (NewHigh > StnLow) THEN
			D[3500 + n] = NewHigh
			D[3600 + n] = D[997]		;Test-Weight
		ENDIF
		D[996] = 0 ;Cancel the Cal-High
	ENDIF

	;Weigh Calculation - Multiply up to give accurate results
	HighLow = StnHigh - StnLow
	HighLow = HighLow * 1000
	;Avoid "Divide By Zero"
	IF (StnTestWgt > 0) THEN
		WeightUnits = DINT(HighLow / StnTestWgt)
		RawLow = INT(StnRaw[n] - StnLow)
		RawLow = RawLow * 1000
		IF (WeightUnits > 0) THEN ;AND (RawLow > 0) THEN
			Stn[n].Weight = INT(RawLow / WeightUnits)
		ELSE
			Stn[n].Weight = 0
		ENDIF
	ELSE
		Stn[n].Weight = 999
	ENDIF

ENDLOOP

IF test THEN
Stn[1].Weight = w1
Stn[2].Weight = w2
Stn[3].Weight = w3
Stn[4].Weight = w4
ENDIF
END_PROGRAM
```

#### zzweigh.var
```iecst
VAR RETAIN
	n : UINT;
	WeightUnits : DINT;
	StnHigh : UINT;
	StnLow : UINT;
	StnTestWgt : UINT;
	HighLow : UDINT;
	RawLow : DINT;
	StnRaw : ARRAY[0..99] OF UINT;
	NewLow : UINT;
	NewHigh : UINT;
END_VAR
VAR
	tstRaw : DINT;
	myRaw : DINT;
	myStnRaw : UINT;
	test : BOOL;
	w1 : UINT;
	w2 : UINT;
	w3 : UINT;
	w4 : UINT;
END_VAR
```

### Program Logical/zztime (IEC) - * System running time

#### zztimeCyclic.ab
```automation-basic
PROGRAM _CYCLIC
(* cyclic program *)

;-------------------
;System Running Time
;-------------------

;-----------------------------------------
;Revision 1.00 12/10/2005 D.J. First Issue
;-----------------------------------------

;Detection of system running - once the detection sequence has remained idle for a given
;period the clock is stopped and the idle time (minutes) is given back. If the idle time
;is 5 minutes and the system stopped at 12:01 then when the time is given back the time will
;read 12:-04 as the time is only taken from the minutes and no the hours count.

;Only use one sequence for system running. Norrmally Offgoing or a loop use the Discharger
D[905]	;Monitor

SystemAction = FALSE
IF D[905] <> Seq THEN
	SystemAction 	= TRUE
	Seq 			= D[905]
ENDIF

R_TRIG(SystemAction,ActionPLS)

TimeNow = clock_ms()

;System Start / Stop Running
IF ActionPLS THEN
	SysRunning 	= TRUE
ENDIF

SysIdleMinutes = 5

TON_10ms(NOT SystemAction,(SysIdleMinutes * 6000),NoAction,NoActionET)

;Read from Graphics
;Seconds = D[310]
Minutes = INT(D[311]) ;Can go minus
Hours	= D[312]

R_TRIG(NoAction,NoActionPLS)

;System has stopped give back the running timer time
IF NoActionPLS THEN
	Minutes 	= Minutes - SysIdleMinutes
	SysRunning 	= FALSE
ENDIF

IF TEST THEN
	Minutes 	= Minutes - 10
	TEST 		= FALSE
ENDIF

IF SysRunning THEN
	TimeDiff	= DiffT(TimeNow,TimeLast)
	MiliSeconds = MiliSeconds + UINT(TimeDiff)
ENDIF

TimeLast = TimeNow

;Count Seconds Running
IF MiliSeconds >= 1000 THEN
	Seconds 	= Seconds + 1
	MiliSeconds = MiliSeconds - 1000 ;Keep and remaing ms to be added next time
ENDIF

IF Seconds >= 60 THEN
	Minutes 	= Minutes + 1
	Seconds 	= Seconds - 60
ENDIF

IF Minutes >= 60 THEN
	Hours 		= Hours + 1
	Minutes	 	= Minutes - 60
ENDIF

;Count Each 1000 hours
IF Hours >= 1000 THEN
	D[313] 		= D[313] + 1
	Hours 		= Hours - 1000
ENDIF

;Store to Graphics
;D[310] = Seconds - don't display seconds as causes TCP/IP driver to send data to Graphics
D[311] = UINT(Minutes)
D[312] = Hours
D[313] = D[313] ;Hours * 1000

END_PROGRAM
```

### Package Logical/Mewa - Your Project Rename

### Package Logical/Mewa/200ms - 200ms Tasks

### can.var
```iecst
VAR
	Box : ARRAY[0..10] OF CAN_Vars;
	CAN : ARRAY[0..32] OF CAN_Vars;
END_VAR
```

### can_cmd.dat
```
;-----------------
;CAN Command Table
;-----------------

;----------------------------------------------------------------------------------------
;Version 2.00 16/08/2011 D.J. Added task name to variables required by AR 3.xx and higher
;----------------------------------------------------------------------------------------

;         1234567890123456789012345678901   1234567890123456789012345678901
00000231,"can_drv2:ReadFrame1            ","can_drv2:EventRead1            ",$00000000
00000230,"can_drv2:WriteFrame1           ","can_drv2:EventWrite1           ",$00000001

;00000131,"can_drv2:ReadFrame2            ","can_drv2:EventRead2            ",$00000000
;00000130,"can_drv2:WriteFrame2           ","can_drv2:EventWrite2           ",$00000001

;00000141,"can_drv2:ReadFrame3            ","can_drv2:EventRead3            ",$00000000
;00000140,"can_drv2:WriteFrame3           ","can_drv2:EventWrite3           ",$00000001
;   |          |                                 |                               |
; CAN ADR  Variable Name 31 Chrs             Event Variable 31 Chrs           Read = 0 Write = 1
```

### Program Logical/Mewa/200ms/CAN/can_drv2 (IEC, version 2.00.0)

#### can_drv2.var
```iecst
VAR RETAIN
	CAN_enable : BOOL;
	ReadFrame1 : WET_CAN;
	EventRead1 : BOOL;
	EventWrite1 : BOOL;
	LastError : UINT;
	n : UINT;
	CANOK : BOOL;
	WriteFrame1 : WET_CAN;
	EventRead2 : BOOL;
	ReadFrame2 : WET_CAN;
	EventWrite2 : BOOL;
	WriteFrame2 : WET_CAN;
END_VAR
VAR
	CANopen_01 : CANopen;
	DOInfo : DatObjInfo;
	CANdftab_01 : CANdftab;
	error_var : UDINT;
	data_adr : UDINT;
	CANrwtab_01 : CANrwtab;
	Remainder : UINT;
	WgtRound : UINT;
END_VAR
```

#### can_drv2.ab
```automation-basic
;CAN Bus data exchange with CBW

;--------------------------------------------------------
;Version 1.00 02/11/2009 D.J. First Issue
;Version 2.00 22/04/2011 D.J. Weight Calculation now here
;--------------------------------------------------------

PROGRAM _INIT

CAN_enable = 1
EventWrite1 = 0									;Reset CAN data table WRITE event
EventRead1 = 0  								;Reset CAN data table READ event
EventWrite2 = 0									;Reset CAN data table WRITE event
EventRead2 = 0  								;Reset CAN data table READ event
;EventWrite3 = 0									;Reset CAN data table WRITE event
;EventRead3 = 0  							    ;Reset CAN data table READ event

CANopen_01.enable		= CAN_enable
CANopen_01.baud_rate	= 25					;Define baud rate - 250 kbit/s
CANopen_01.cob_anz		= 100      				;Define number of link objects
CANopen_01.error_adr	= ADR(error_var)		;Define address for error output
CANopen_01.device		= ADR("SL1.IF1.ST1.IF1.ST2.IF1")	;Define number of device
CANopen_01.info			= 0

CANopen_01 FUB CANopen()						;Initiate CANopen

IF CANopen_01.status=0 THEN						;Check error level

	DOInfo.enable = 1
	DOInfo.pName  = "can_cmd"

	DOInfo FUB DatObjInfo()

	IF (DOInfo.status = 0) THEN

		data_adr					= DOInfo.pDatObjMem
		CANdftab_01.enable			= 1
		CANdftab_01.us_ident 		= CANopen_01.us_ident	;Set us_id
		CANdftab_01.table_adr		= data_adr				;Define address of data object
		CANdftab_01.tab_num			= UINT(DOInfo.len / 72)	;Define number of values

		CANdftab_01 FUB CANdftab()    						;Initiate CANdftab

		IF CANdftab_01.status = 0 THEN
			WriteFrame1.ControlSignals = BIT_SET(WriteFrame1.ControlSignals,0);Set Live Signal
			;WriteFrame2.ControlSignals = BIT_SET(WriteFrame2.ControlSignals,0)
			;WriteFrame3.ControlSignals = BIT_SET(WriteFrame3.ControlSignals,0)
			CANOK = TRUE
		ENDIF

	ENDIF

ENDIF

END_PROGRAM

PROGRAM _CYCLIC

IF CANOK THEN

	;----------------
	;Set Write values
	;----------------

	;------------------------------------------------------
	;Configure the CAN write to CBW1 SDC1
	;------------------------------------------------------
Line[7].SpaceBIT
	IF (Line[7].SpaceBIT>0) AND CAN[1].BagReady THEN
		WriteFrame1.ControlSignals = BIT_SET(WriteFrame1.ControlSignals, 1)
	ELSE
		WriteFrame1.ControlSignals = BIT_CLR(WriteFrame1.ControlSignals, 1)
	ENDIF
	IF (Line[5].SpaceBIT>0) AND CAN[1].BagReady THEN
		WriteFrame1.ControlSignals = BIT_SET(WriteFrame1.ControlSignals, 2)
	ELSE
		WriteFrame1.ControlSignals = BIT_CLR(WriteFrame1.ControlSignals, 2)
	ENDIF
	EventWrite1 = TRUE

	;WriteFrame1.FaultNumber = 0
	WriteFrame1.Category = 0
	WriteFrame1.Customer    = 0
	WriteFrame1.Weight      = 0

	;------------------------
	;Service CAN table
	;------------------------

	IF CANdftab_01.status=0 THEN						(*check error level*)
		CANrwtab_01.enable		= 1
		CANrwtab_01.tab_ident	= CANdftab_01.tab_ident (*define tab_id*)
		CANrwtab_01 FUB CANrwtab()						(*initiate CANrwtab*)
		LastError = CANrwtab_01.status
	ENDIF

	;----------------------------------------------------
	;Check for incomming data from CBW1
	;----------------------------------------------------
	IF EventRead1 THEN
		EventRead1 = FALSE

		CAN[1].Live 			= BIT_TST(ReadFrame1.ControlSignals,0)
		CAN[1].UnloadFinished 	= BIT_TST(ReadFrame1.ControlSignals,1)
	;	CAN[1].FaultNumber		= ReadFrame1.FaultNumber
		CAN[1].Category			= ReadFrame1.Category
		CAN[1].Customer			= ReadFrame1.Customer
		CAN[1].Weight			= ReadFrame1.Weight

		IF CAN[1].Live THEN
			CAN[1].LiveTime = 50	;5 seconds
		ENDIF
	ENDIF

	IF NOT CAN[1].Live THEN
		ReadFrame1.ControlSignals = BIT_CLR(ReadFrame1.ControlSignals,0)
	ENDIF

	;-----------------
	;Live section
	;-----------------
	LOOP n = 1 TO 8 DO
		IF (CAN[n].LiveTime > 0) THEN
			CAN[n].LiveTime = (CAN[n].LiveTime - 1)
		ENDIF
		CAN[n].Live = (CAN[n].LiveTime <> 0)
	ENDLOOP
ENDIF

;Monitor Registers for TrackView
D[91] = UINT(ReadFrame1.ControlSignals)	;ID = 231
D[92] = UINT(WriteFrame1.ControlSignals);ID = 230

END_PROGRAM
```

### can_live.var
```iecst
VAR
	CANLive_1	:BIT_ENCODE;
	CANLive_2	:BIT_ENCODE;
END_VAR
```

### can_stn.var
```iecst
VAR RETAIN
	CAN_enable : BOOL;
	LastError : UINT;
	n : UINT;
	CANOK : BOOL;
END_VAR
VAR
	Box1Cust : UINT;
END_VAR
VAR RETAIN
	Box1Cus : UINT;
	Box2Cus : UINT;
	Box3Cus : UINT;
	Box4Cus : UINT;
	Box5Cus : UINT;
	Box6Cus : UINT;
END_VAR
VAR
	WriteFrame1115 : Box_CUS_DST;
	WriteFrame1104 : Box_SP_CAT;
	WriteFrame1105 : Box_SP_CAT;
	WriteFrame1114 : Box_CUS_DST;
	WriteFrame1102 : Box_SP_CAT;
	WriteFrame1101 : Box_SP_CAT;
	WriteFrame1113 : Box_CUS_DST;
	WriteFrame1103 : Box_SP_CAT;
	WriteFrame1112 : Box_CUS_DST;
	WriteFrame1111 : Box_CUS_DST;
	CANopen_01 : CANopen;
	DOInfo : DatObjInfo;
	CANdftab_01 : CANdftab;
	error_var : UDINT;
	CANrwtab_01 : CANrwtab;
	EventRead1001 : BOOL;
	EventRead1011 : BOOL;
	EventWrite1021 : BOOL;
	EventWrite1101 : BOOL;
	EventWrite1111 : BOOL;
	EventRead1002 : BOOL;
	EventRead1012 : BOOL;
	EventWrite1022 : BOOL;
	EventWrite1102 : BOOL;
	EventWrite1112 : BOOL;
	EventRead1003 : BOOL;
	EventRead1013 : BOOL;
	EventWrite1023 : BOOL;
	EventWrite1103 : BOOL;
	EventWrite1113 : BOOL;
	EventRead1004 : BOOL;
	EventRead1014 : BOOL;
	EventWrite1024 : BOOL;
	EventWrite1104 : BOOL;
	EventWrite1114 : BOOL;
	EventRead1005 : BOOL;
	EventRead1015 : BOOL;
	EventWrite1025 : BOOL;
	EventWrite1105 : BOOL;
	EventWrite1115 : BOOL;
	EventRead1006 : BOOL;
	EventRead1016 : BOOL;
	EventWrite1026 : BOOL;
	EventWrite1106 : BOOL;
	EventWrite1116 : BOOL;
	EventRead1007 : BOOL;
	EventRead1017 : BOOL;
	EventWrite1027 : BOOL;
	EventWrite1107 : BOOL;
	EventWrite1117 : BOOL;
	EventRead1008 : BOOL;
	EventRead1018 : BOOL;
	EventWrite1028 : BOOL;
	EventWrite1108 : BOOL;
	EventWrite1118 : BOOL;
	EventRead1009 : BOOL;
	EventRead1019 : BOOL;
	EventWrite1029 : BOOL;
	EventWrite1109 : BOOL;
	EventWrite1119 : BOOL;
	WriteFrame1026 : WET_CAN;
	WriteFrame1025 : WET_CAN;
	WriteFrame1024 : WET_CAN;
	WriteFrame1023 : WET_CAN;
	WriteFrame1021 : WET_CAN;
	WriteFrame1022 : WET_CAN;
	WriteFrame1027 : WET_CAN;
	WriteFrame1028 : WET_CAN;
	WriteFrame1029 : WET_CAN;
	WriteFrame1106 : Box_SP_CAT;
	WriteFrame1107 : Box_SP_CAT;
	WriteFrame1108 : Box_SP_CAT;
	WriteFrame1109 : Box_SP_CAT;
	WriteFrame1116 : Box_CUS_DST;
	WriteFrame1117 : Box_CUS_DST;
	WriteFrame1118 : Box_CUS_DST;
	WriteFrame1119 : Box_CUS_DST;
	TimeNow : TIME;
	TimeLastWrite : TIME;
	WriteEvent : BOOL;
	DatabaseChanged : UINT;
	wTabNum : UINT;
	strName_can_tab : ARRAY[0..9] OF USINT;
	TimeDiff : UINT;
	ReadFrame1001 : Box_CUS_BAT;
	ReadFrame1002 : Box_CUS_BAT;
	ReadFrame1003 : Box_CUS_BAT;
	ReadFrame1004 : Box_CUS_BAT;
	ReadFrame1005 : Box_CUS_BAT;
	ReadFrame1006 : Box_CUS_BAT;
	ReadFrame1007 : Box_CUS_BAT;
	ReadFrame1008 : Box_CUS_BAT;
	ReadFrame1009 : Box_CUS_BAT;
	Dummy : UDINT;
	ReadFrame1011 : Box_CONTROL;
	ReadFrame1012 : Box_CONTROL;
	ReadFrame1013 : Box_CONTROL;
	ReadFrame1014 : Box_CONTROL;
	ReadFrame1015 : Box_CONTROL;
	ReadFrame1016 : Box_CONTROL;
	ReadFrame1017 : Box_CONTROL;
	ReadFrame1018 : Box_CONTROL;
	ReadFrame1019 : Box_CONTROL;
	t : UINT;
END_VAR
```

### can_stns.dat
```
;-----------------
;CAN Command Table
;-----------------

;         1234567890123446789012344678901   1234567890123446789012344678901
;Box 1
00001001,"can_stn:ReadFrame1001          ","can_stn:EventRead1001          ",$00000000
00001011,"can_stn:ReadFrame1011          ","can_stn:EventRead1011          ",$00000000
00001021,"can_stn:WriteFrame1021         ","can_stn:EventWrite1021         ",$00000001
00001101,"can_stn:WriteFrame1101         ","can_stn:EventWrite1101         ",$00000001
00001111,"can_stn:WriteFrame1111         ","can_stn:EventWrite1111         ",$00000001

;Box 2
00001002,"can_stn:ReadFrame1002          ","can_stn:EventRead1002          ",$00000000
00001012,"can_stn:ReadFrame1012          ","can_stn:EventRead1012          ",$00000000
00001022,"can_stn:WriteFrame1022         ","can_stn:EventWrite1022         ",$00000001
00001102,"can_stn:WriteFrame1102         ","can_stn:EventWrite1102         ",$00000001
00001112,"can_stn:WriteFrame1112         ","can_stn:EventWrite1112         ",$00000001

;Box 3
00001003,"can_stn:ReadFrame1003          ","can_stn:EventRead1003          ",$00000000
00001013,"can_stn:ReadFrame1013          ","can_stn:EventRead1013          ",$00000000
00001023,"can_stn:WriteFrame1023         ","can_stn:EventWrite1023         ",$00000001
00001103,"can_stn:WriteFrame1103         ","can_stn:EventWrite1103         ",$00000001
00001113,"can_stn:WriteFrame1113         ","can_stn:EventWrite1113         ",$00000001

;Box 4
00001004,"can_stn:ReadFrame1004          ","can_stn:EventRead1004          ",$00000000
00001014,"can_stn:ReadFrame1014          ","can_stn:EventRead1014          ",$00000000
00001024,"can_stn:WriteFrame1024         ","can_stn:EventWrite1024         ",$00000001
00001104,"can_stn:WriteFrame1104         ","can_stn:EventWrite1104         ",$00000001
00001114,"can_stn:WriteFrame1114         ","can_stn:EventWrite1114         ",$00000001

;Box 5
00001005,"can_stn:ReadFrame1005          ","can_stn:EventRead1005          ",$00000000
00001015,"can_stn:ReadFrame1015          ","can_stn:EventRead1015          ",$00000000
00001025,"can_stn:WriteFrame1025         ","can_stn:EventWrite1025         ",$00000001
00001105,"can_stn:WriteFrame1105         ","can_stn:EventWrite1105         ",$00000001
00001115,"can_stn:WriteFrame1115         ","can_stn:EventWrite1115         ",$00000001

;Box 6
00001006,"can_stn:ReadFrame1006          ","can_stn:EventRead1006          ",$00000000
00001016,"can_stn:ReadFrame1016          ","can_stn:EventRead1016          ",$00000000
00001026,"can_stn:WriteFrame1026         ","can_stn:EventWrite1026         ",$00000001
00001106,"can_stn:WriteFrame1106         ","can_stn:EventWrite1106         ",$00000001
00001116,"can_stn:WriteFrame1116         ","can_stn:EventWrite1116         ",$00000001

;Box 7
00001007,"can_stn:ReadFrame1007          ","can_stn:EventRead1007          ",$00000000
00001017,"can_stn:ReadFrame1017          ","can_stn:EventRead1017          ",$00000000
00001027,"can_stn:WriteFrame1027         ","can_stn:EventWrite1027         ",$00000001
00001107,"can_stn:WriteFrame1107         ","can_stn:EventWrite1107         ",$00000001
00001117,"can_stn:WriteFrame1117         ","can_stn:EventWrite1117         ",$00000001

;Box 8
00001008,"can_stn:ReadFrame1008          ","can_stn:EventRead1008          ",$00000000
00001018,"can_stn:ReadFrame1018          ","can_stn:EventRead1018          ",$00000000
00001028,"can_stn:WriteFrame1028         ","can_stn:EventWrite1028         ",$00000001
00001108,"can_stn:WriteFrame1108         ","can_stn:EventWrite1108         ",$00000001
00001118,"can_stn:WriteFrame1118         ","can_stn:EventWrite1118         ",$00000001

;Box 9
00001009,"can_stn:ReadFrame1009          ","can_stn:EventRead1009          ",$00000000
00001019,"can_stn:ReadFrame1019          ","can_stn:EventRead1019          ",$00000000
00001029,"can_stn:WriteFrame1029         ","can_stn:EventWrite1029         ",$00000001
00001109,"can_stn:WriteFrame1109         ","can_stn:EventWrite1109         ",$00000001
00001119,"can_stn:WriteFrame1119         ","can_stn:EventWrite1119         ",$00000001

;   |          |                                 |                               |
; CAN ADR  Variable Name 31 Chrs             Event Variable 31 Chrs           Read = 0 Write = 1
```

Listed in the project but not available here: Logical/Reference/5_ppf1, Logical/Reference/8_pwb3/pwb.var, Logical/Reference/12_pup4, Logical/Reference/15_pbr1/pbr.ab, Logical/Reference/15_pbr1/pbr.var, Logical/Reference/31_picu13, Logical/Reference/32_picd3, Logical/Reference/35_picu6, Logical/Reference/37_picu8, Logical/Reference/40_picu11, Logical/Reference/41_picd12, Logical/Reference/43_picd14, Logical/Reference/45_picu16, Logical/Reference/46_picu17, Logical/Reference/50_fb_pr, Logical/Sequences/10ms/zzStnSer/zzstnser.var, Logical/Sequences/10ms/zzCount/zzcount.var, Logical/Sequences/10ms/zzStnMix/zzstnmix.var, Logical/Sequences/10ms/1_clu_1/3_slu_1Init.ab, Logical/Sequences/10ms/3_slu_1/3_slu_1Init.ab, Logical/Sequences/10ms/10_sdc5/6_sdc1Init.ab, Logical/Sequences/10ms/14_cvc2/8_svc1Init.ab, Logical/Sequences/10ms/20_cpc1/9_spc1Init.ab, Logical/Sequences/10ms/22_cic7/9_spc1Init.ab, Logical/Sequences/10ms/24_csb1/7_svc1Init.ab, Logical/Sequences/10ms/25_cp16/10_bsonInit.ab, Logical/Sequences/10ms/27_csb2/12_svc2Init.ab, Logical/Sequences/10ms/zzAI2744/zzAI2744.var, Logical/Sequences/10ms/zzIndi/zzindi.var, Logical/Sequences/10ms/zzIndi/zzindiCyclic.ab, Logical/Sequences/10ms/zzTCPIP/zztcpip.var, Logical/Sequences/10ms/zzTCPIP/zztcpip.ab, Logical/Sequences/10ms/zzIO/zzio.var, Logical/Sequences/200ms/udp_CTT/udp_CTT.var, Logical/Sequences/200ms/udp_CTT/UDP_CTT, Logical/Sequences/200ms/USB_Pmem/usb_pmem.var, Logical/Sequences/200ms/zzAlarms/zzalarms.var, Logical/Sequences/200ms/zzAlarms/zzalarms.ab, Logical/Sequences/TB/12_belt2/12_belt2.var, Logical/Sequences/TB/12_belt2/12_belt2.ab, Logical/Sequences/zzalarms/zzalarmsInit.ab, Logical/Sequences/zzclrmem/zzclrmem.var, Logical/Sequences/zzclrmem/zzclrmemInit.ab, Logical/Sequences/zzclrmem/zzclrmemCyclic.ab, Logical/Sequences/zzconst/zzconst.var, Logical/Sequences/zzindi/zzindiInit.ab, Logical/Sequences/zzindi/zzindiCyclic.ab, Logical/Sequences/zzio/zzioInit.ab, Logical/Sequences/zzreport/zzreport.var, Logical/Sequences/zzreport/zzreportInit.ab, Logical/Sequences/zzreport/zzreportCyclic.ab, Logical/Sequences/zzstd/zzstd.var, Logical/Sequences/zzstd/zzstdInit.ab, Logical/Sequences/zzstd/zzstdCyclic.ab, Logical/Sequences/zztc2end/zztc2end.var, Logical/Sequences/zztc2end/zztc2endInit.ab, Logical/Sequences/zztcpip/zztcpip.var, Logical/Sequences/zztcpip/zztcpipInit.ab, Logical/Sequences/zztrip/zztrip.var, Logical/Sequences/zztrip/zztripInit.ab, Logical/Libraries/SupLib4/SupLib4.fun, Logical/Libraries/SupLib4/BCD_BIN_OUTPUT.ab, Logical/Libraries/SupLib4/BIN_TO_BCD.ab, Logical/Libraries/SupLib4/BIT_ENCODE.ab, Logical/Libraries/SupLib4/DIS4.ab, Logical/Libraries/SupLib4/stASC_UINT.ab, Logical/Libraries/SupLib4/stUINT_ASC.ab, Logical/Libraries/SupLib4/stUNI4.ab, Logical/Libraries/SupLib4/stUNI5.ab, Logical/Libraries/WETCAN2/WETCAN2.typ, Logical/Libraries/WETCAN2/CAN2Init.ab, Logical/Libraries/WETCAN2/_SetCAN1TypeToByteArray.ab, Logical/Libraries/WETCAN2/_version.ab, Logical/Libraries/WETCAN2/_Seti386CAN2TypeToCAN1Type.ab, Logical/Libraries/WETCAN2/_swapUINT.ab, Logical/Libraries/WETCAN2/WETCAN2.fun, Logical/Timestamp/Timestamp.typ, Logical/Timestamp/zzGetTime, Logical/SQL/SQL.typ, Logical/SQL/zzTvText/zzTvText.typ, Logical/SQL/zzTvText/zzTvText.var, Logical/SQL/zzSQL_Lib/zzSQL_Lib.typ, Logical/SQL/zzSQL_Lib/zzSQL_Lib.var, Logical/SQL/zzSQL_Lib/Constants.var, Logical/SQL/SQLSpeedTest/SQLSpeedTestCyclic.ab, Logical/SQL/zzGetNamesSQL/zzGetNameSQL.typ, Logical/SQL/zzGetNamesSQL/zzGetNameSQL.var, Logical/SQL/zzGetNamesSQL/zzGetNameSQL/zzGetNames.var, Logical/SQL/zzGetNamesSQL/zzGetNameSQL/zzGetNames.ab, Logical/SQL/Test_bagMaint/Test_bagMaint.var, Logical/zztc2end, Logical/zzclrmem/zzclrmemCyclic.ab, Logical/zzclrmem/zzclrmemInit.ab, Logical/zzclrmem/zzclrmem.var, Logical/zzweigh/zzweighInit.ab, Logical/zzreport
